// TIA Portal V17 export
// export: Created 2023-02-13T11:16:34.9023013Z, ExportSetting WithDefaults, DisplayName Totally Integrated Automation Portal, DisplayVersion V17, DisplayName TIA Portal Openness, DisplayVersion V17, DisplayName TIA Portal Teamcenter Gateway, DisplayVersion V17, DisplayName TIA Portal Version Control Interface, DisplayVersion V17, DisplayName SINAMICS Startdrive Advanced, DisplayVersion V17, DisplayName SINAMICS Startdrive G130, G150, S120, S150, SINAMICS MV, S210, DisplayVersion V17, DisplayName SINAMICS Startdrive G110M, G120, G120C, G120D, G120P, G115D, DisplayVersion V17, DisplayName STEP 7 Professional, DisplayVersion V17, DisplayName STEP 7 Safety, DisplayVersion V17, DisplayName WinCC Professional, DisplayVersion V17
FUNCTION_BLOCK "IO_Valve_Buffer"   // FB19, LAD
{ S7_Optimized_Access := 'FALSE' }
VERSION : 0.1
// stored: AutoNumber true, IsIECCheckEnabled false, SetENOAutomatically false, UDAEnableTagReadback false
   VAR_INPUT
      "lock 1" : Bool;
      "lock 2" : Bool;
      "lock 3" : Bool;
      "lock 4" : Bool;
      init : Bool;
      reset : Bool;
      testing : Bool;
   END_VAR
   VAR
      "AV-22.11" : "Valve";
      "AV-22.21" : "Valve";
      "AV-22.22" : "Valve";
      "AV-22.23" : "Valve";
      "AV-32.01" : "Valve";
      "AV-32.02" : "Valve";
      "AV-32.03" : "Valve";
      "AV-32.04" : "Valve";
      "AV-32.11" : "Valve";
      "AV-32.21" : "Valve";
      "AV-32.22" : "Valve";
      "AV-32.23" : "Valve";
      "AV-61.01" : "Valve";
      "AV-61.02" : "Valve";
      "AV-61.03" : "Valve";
      "AV-61.04" : "Valve";
      "AV-61.05" : "Valve";
      "AV-61.21" : "Valve";
      "AV-62.06" : "Valve";
      "AV-64.01" : "Valve";
      "AV-64.02" : "Valve";
      "AV-64.03" : "Valve";
      "AV-64.04" : "Valve";
      "AV-64.05" : "Valve";
      "AV-64.06" : "Valve";
      "AV-65.01" : "Valve";
      "AV-65.02" : "Valve";
      "AV-65.03" : "Valve";
      "AV-65.04" : "Valve";
      "AV-65.05" : "Valve";
      "AV-65.21" : "Valve";
      "AV-66.01" : "Valve";
      "AV-66.02" : "Valve";
      "AV-66.03" : "Valve";
      "AV-66.04" : "Valve";
      "AV-66.05" : "Valve";
      "AV-66.06" : "Valve";
      "AV-67.01" : "Valve";
      "AV-67.02" : "Valve";
      "AV-67.03" : "Valve";
      "AV-67.04" : "Valve";
      "AV-67.05" : "Valve";
      "AV-68.01" : "Valve";
      "AV-68.02" : "Valve";
      "AV-68.03" : "Valve";
      "AV-68.04" : "Valve";
      "AV-68.05" : "Valve";
      "AV-68.06" : "Valve";
   END_VAR
BEGIN

REGION Network 1 (SCL): FB OPEN AND CLOSE VALVE T-22
   IF #testing THEN
       // Statement section IF
       #"AV-22.11".FB_OPEN := #"AV-22.11".QCMD_OP;
       #"AV-22.11".FB_CLOSE := NOT #"AV-22.11".QCMD_OP;
       #"AV-22.21".FB_OPEN := #"AV-22.21".QCMD_OP;
       #"AV-22.21".FB_CLOSE := NOT #"AV-22.21".QCMD_OP;
       #"AV-22.22".FB_OPEN := #"AV-22.22".QCMD_OP;
       #"AV-22.22".FB_CLOSE := NOT #"AV-22.22".QCMD_OP;
       #"AV-22.23".FB_OPEN := #"AV-22.23".QCMD_OP;
       #"AV-22.23".FB_CLOSE := NOT #"AV-22.23".QCMD_OP;
   ELSE
       // Statement section ELSE
       #"AV-22.11".FB_OPEN := #"AV-22.11".QCMD_OP;
       #"AV-22.11".FB_CLOSE := NOT #"AV-22.11".QCMD_OP;
       #"AV-22.21".FB_OPEN := #"AV-22.21".QCMD_OP;
       #"AV-22.21".FB_CLOSE := NOT #"AV-22.21".QCMD_OP;
       #"AV-22.22".FB_OPEN := #"AV-22.22".QCMD_OP;
       #"AV-22.22".FB_CLOSE := NOT #"AV-22.22".QCMD_OP;
       #"AV-22.23".FB_OPEN := #"AV-22.23".QCMD_OP;
       #"AV-22.23".FB_CLOSE := NOT #"AV-22.23".QCMD_OP;
   END_IF;
END_REGION

NETWORK
TITLE = FB MONITORING TIME VALVE T-22
// FB OPEN TIME
      L     T#20s;
      T     #"AV-22.11".MON_T;
      T     #"AV-22.21".MON_T;
      T     #"AV-22.22".MON_T;
      T     #"AV-22.23".MON_T;
// FB CLOSE TIME
      L     T#20s;
      T     #"AV-22.11".MON_T_CLOSE;
      T     #"AV-22.21".MON_T_CLOSE;
      T     #"AV-22.22".MON_T_CLOSE;
      T     #"AV-22.23".MON_T_CLOSE;


REGION Network 3: AV-22.11
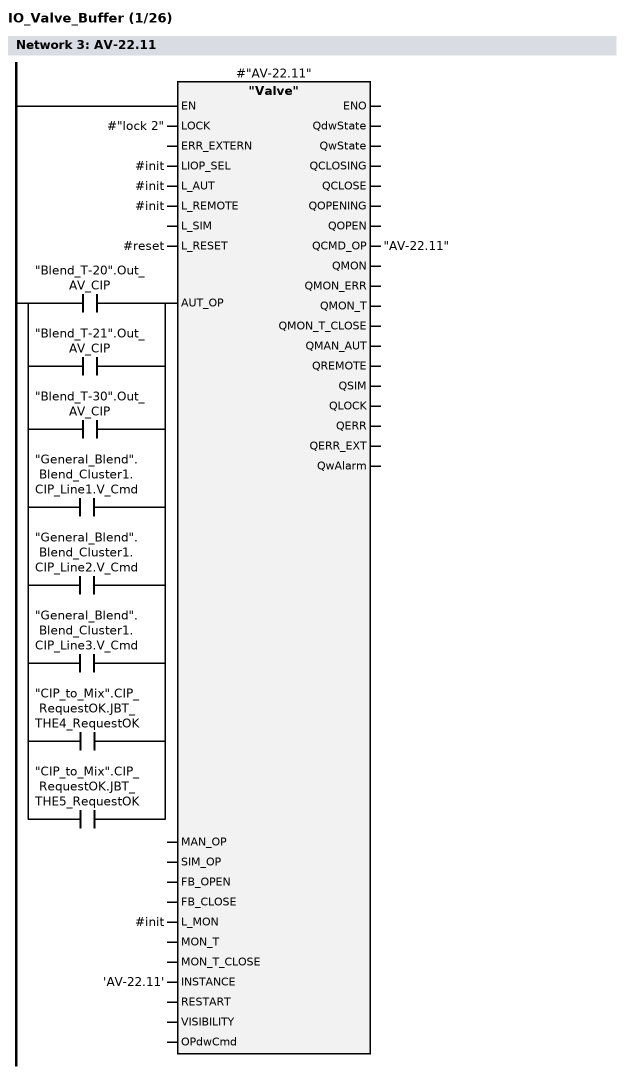
   RUNG wire#powerrail
      #"AV-22.11"(AUT_OP := wire#w1, LOCK := #"lock 2", ERR_EXTERN :=, LIOP_SEL := #init, L_AUT := #init, L_REMOTE := #init, L_SIM :=, L_RESET := #reset, MAN_OP :=, SIM_OP :=, FB_OPEN :=, FB_CLOSE :=, L_MON := #init, MON_T :=, MON_T_CLOSE :=, INSTANCE := 'AV-22.11', RESTART :=, VISIBILITY :=, OPdwCmd :=, QdwState =>, QwState =>, QCLOSING =>, QCLOSE =>, QOPENING =>, QOPEN =>, QCMD_OP => "AV-22.11", QMON =>, QMON_ERR =>, QMON_T =>, QMON_T_CLOSE =>, QMAN_AUT =>, QREMOTE =>, QSIM =>, QLOCK =>, QERR =>, QERR_EXT =>, QwAlarm =>)
   END_RUNG
   RUNG wire#powerrail
      Contact( "Blend_T-20".Out_AV_CIP )
   END_RUNG wire#w1
   RUNG wire#powerrail
      Contact( "Blend_T-21".Out_AV_CIP )
   END_RUNG wire#w1
   RUNG wire#powerrail
      Contact( "Blend_T-30".Out_AV_CIP )
   END_RUNG wire#w1
   RUNG wire#powerrail
      Contact( "General_Blend".Blend_Cluster1.CIP_Line1.V_Cmd )
   END_RUNG wire#w1
   RUNG wire#powerrail
      Contact( "General_Blend".Blend_Cluster1.CIP_Line2.V_Cmd )
   END_RUNG wire#w1
   RUNG wire#powerrail
      Contact( "General_Blend".Blend_Cluster1.CIP_Line3.V_Cmd )
   END_RUNG wire#w1
   RUNG wire#powerrail
      Contact( "CIP_to_Mix".CIP_RequestOK.JBT_THE4_RequestOK )
   END_RUNG wire#w1
   RUNG wire#powerrail
      Contact( "CIP_to_Mix".CIP_RequestOK.JBT_THE5_RequestOK )
   END_RUNG wire#w1
   // the same network as SCL:
   #"AV-22.11"(LOCK := #"lock 2",   // "Valve"
               LIOP_SEL := #init,
               L_AUT := #init,
               L_REMOTE := #init,
               L_RESET := #reset,
               AUT_OP := "Blend_T-20".Out_AV_CIP OR "Blend_T-21".Out_AV_CIP OR "Blend_T-30".Out_AV_CIP OR "General_Blend".Blend_Cluster1.CIP_Line1.V_Cmd OR "General_Blend".Blend_Cluster1.CIP_Line2.V_Cmd OR "General_Blend".Blend_Cluster1.CIP_Line3.V_Cmd OR "CIP_to_Mix".CIP_RequestOK.JBT_THE4_RequestOK OR "CIP_to_Mix".CIP_RequestOK.JBT_THE5_RequestOK,
               L_MON := #init,
               INSTANCE := 'AV-22.11',
               QCMD_OP => "AV-22.11");
END_REGION

REGION Network 4: AV-22.21
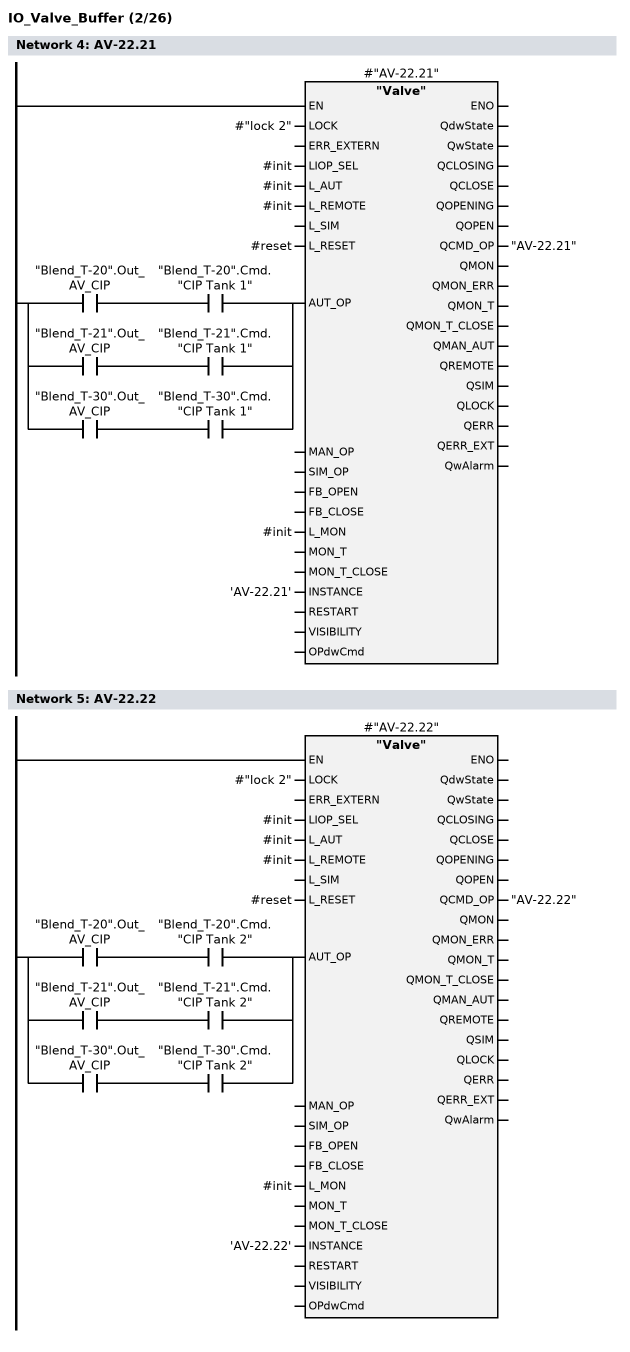
   RUNG wire#powerrail
      #"AV-22.21"(AUT_OP := wire#w1, LOCK := #"lock 2", ERR_EXTERN :=, LIOP_SEL := #init, L_AUT := #init, L_REMOTE := #init, L_SIM :=, L_RESET := #reset, MAN_OP :=, SIM_OP :=, FB_OPEN :=, FB_CLOSE :=, L_MON := #init, MON_T :=, MON_T_CLOSE :=, INSTANCE := 'AV-22.21', RESTART :=, VISIBILITY :=, OPdwCmd :=, QdwState =>, QwState =>, QCLOSING =>, QCLOSE =>, QOPENING =>, QOPEN =>, QCMD_OP => "AV-22.21", QMON =>, QMON_ERR =>, QMON_T =>, QMON_T_CLOSE =>, QMAN_AUT =>, QREMOTE =>, QSIM =>, QLOCK =>, QERR =>, QERR_EXT =>, QwAlarm =>)
   END_RUNG
   RUNG wire#powerrail
      Contact( "Blend_T-20".Out_AV_CIP )
      Contact( "Blend_T-20".Cmd."CIP Tank 1" )
   END_RUNG wire#w1
   RUNG wire#powerrail
      Contact( "Blend_T-21".Out_AV_CIP )
      Contact( "Blend_T-21".Cmd."CIP Tank 1" )
   END_RUNG wire#w1
   RUNG wire#powerrail
      Contact( "Blend_T-30".Out_AV_CIP )
      Contact( "Blend_T-30".Cmd."CIP Tank 1" )
   END_RUNG wire#w1
   // the same network as SCL:
   #"AV-22.21"(LOCK := #"lock 2",   // "Valve"
               LIOP_SEL := #init,
               L_AUT := #init,
               L_REMOTE := #init,
               L_RESET := #reset,
               AUT_OP := ("Blend_T-20".Out_AV_CIP AND "Blend_T-20".Cmd."CIP Tank 1") OR ("Blend_T-21".Out_AV_CIP AND "Blend_T-21".Cmd."CIP Tank 1") OR ("Blend_T-30".Out_AV_CIP AND "Blend_T-30".Cmd."CIP Tank 1"),
               L_MON := #init,
               INSTANCE := 'AV-22.21',
               QCMD_OP => "AV-22.21");
END_REGION

REGION Network 5: AV-22.22
   RUNG wire#powerrail
      #"AV-22.22"(AUT_OP := wire#w1, LOCK := #"lock 2", ERR_EXTERN :=, LIOP_SEL := #init, L_AUT := #init, L_REMOTE := #init, L_SIM :=, L_RESET := #reset, MAN_OP :=, SIM_OP :=, FB_OPEN :=, FB_CLOSE :=, L_MON := #init, MON_T :=, MON_T_CLOSE :=, INSTANCE := 'AV-22.22', RESTART :=, VISIBILITY :=, OPdwCmd :=, QdwState =>, QwState =>, QCLOSING =>, QCLOSE =>, QOPENING =>, QOPEN =>, QCMD_OP => "AV-22.22", QMON =>, QMON_ERR =>, QMON_T =>, QMON_T_CLOSE =>, QMAN_AUT =>, QREMOTE =>, QSIM =>, QLOCK =>, QERR =>, QERR_EXT =>, QwAlarm =>)
   END_RUNG
   RUNG wire#powerrail
      Contact( "Blend_T-20".Out_AV_CIP )
      Contact( "Blend_T-20".Cmd."CIP Tank 2" )
   END_RUNG wire#w1
   RUNG wire#powerrail
      Contact( "Blend_T-21".Out_AV_CIP )
      Contact( "Blend_T-21".Cmd."CIP Tank 2" )
   END_RUNG wire#w1
   RUNG wire#powerrail
      Contact( "Blend_T-30".Out_AV_CIP )
      Contact( "Blend_T-30".Cmd."CIP Tank 2" )
   END_RUNG wire#w1
   // the same network as SCL:
   #"AV-22.22"(LOCK := #"lock 2",   // "Valve"
               LIOP_SEL := #init,
               L_AUT := #init,
               L_REMOTE := #init,
               L_RESET := #reset,
               AUT_OP := ("Blend_T-20".Out_AV_CIP AND "Blend_T-20".Cmd."CIP Tank 2") OR ("Blend_T-21".Out_AV_CIP AND "Blend_T-21".Cmd."CIP Tank 2") OR ("Blend_T-30".Out_AV_CIP AND "Blend_T-30".Cmd."CIP Tank 2"),
               L_MON := #init,
               INSTANCE := 'AV-22.22',
               QCMD_OP => "AV-22.22");
END_REGION

REGION Network 6: AV-22.23
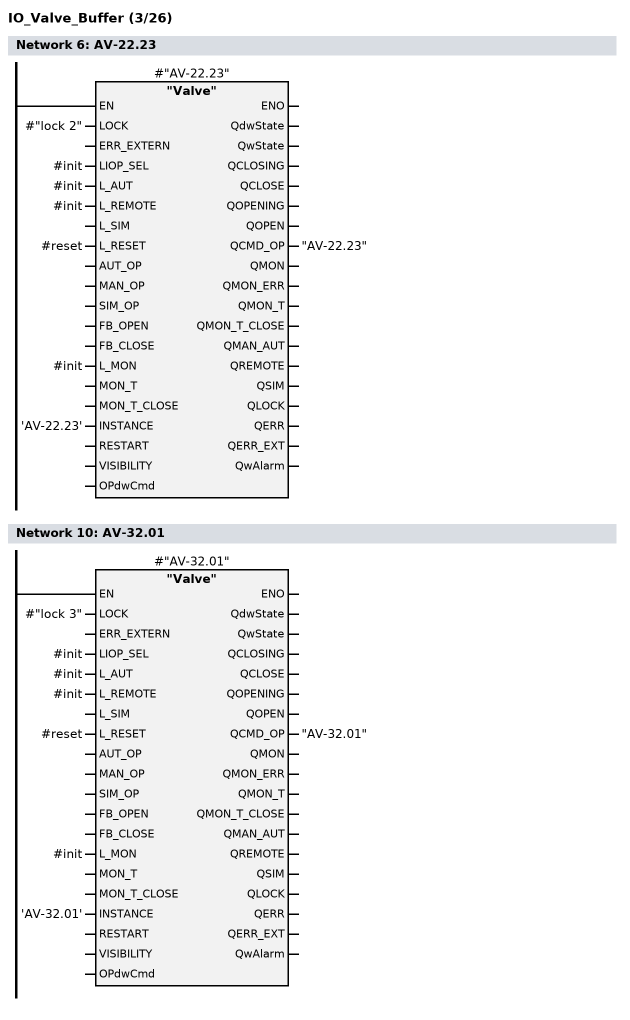
   RUNG wire#powerrail
      #"AV-22.23"(LOCK := #"lock 2", ERR_EXTERN :=, LIOP_SEL := #init, L_AUT := #init, L_REMOTE := #init, L_SIM :=, L_RESET := #reset, AUT_OP :=, MAN_OP :=, SIM_OP :=, FB_OPEN :=, FB_CLOSE :=, L_MON := #init, MON_T :=, MON_T_CLOSE :=, INSTANCE := 'AV-22.23', RESTART :=, VISIBILITY :=, OPdwCmd :=, QdwState =>, QwState =>, QCLOSING =>, QCLOSE =>, QOPENING =>, QOPEN =>, QCMD_OP => "AV-22.23", QMON =>, QMON_ERR =>, QMON_T =>, QMON_T_CLOSE =>, QMAN_AUT =>, QREMOTE =>, QSIM =>, QLOCK =>, QERR =>, QERR_EXT =>, QwAlarm =>)
   END_RUNG
   // the same network as SCL:
   #"AV-22.23"(LOCK := #"lock 2",   // "Valve"
               LIOP_SEL := #init,
               L_AUT := #init,
               L_REMOTE := #init,
               L_RESET := #reset,
               L_MON := #init,
               INSTANCE := 'AV-22.23',
               QCMD_OP => "AV-22.23");
END_REGION

REGION Network 8 (SCL): FB OPEN AND CLOSE VALVE T-32
   IF #testing THEN
       // Statement section IF
       #"AV-32.01".FB_OPEN := #"AV-32.01".QCMD_OP;
       #"AV-32.01".FB_CLOSE := NOT #"AV-32.01".QCMD_OP;
       #"AV-32.02".FB_OPEN := #"AV-32.02".QCMD_OP;
       #"AV-32.02".FB_CLOSE := NOT #"AV-32.02".QCMD_OP;
       #"AV-32.03".FB_OPEN := #"AV-32.03".QCMD_OP;
       #"AV-32.03".FB_CLOSE := NOT #"AV-32.03".QCMD_OP;
       #"AV-32.04".FB_OPEN := #"AV-32.04".QCMD_OP;
       #"AV-32.04".FB_CLOSE := NOT #"AV-32.04".QCMD_OP;
       #"AV-32.11".FB_OPEN := #"AV-32.11".QCMD_OP;
       #"AV-32.11".FB_CLOSE := NOT #"AV-32.11".QCMD_OP;
       #"AV-32.21".FB_OPEN := #"AV-32.21".QCMD_OP;
       #"AV-32.21".FB_CLOSE := NOT #"AV-32.21".QCMD_OP;
       #"AV-32.22".FB_OPEN := #"AV-32.22".QCMD_OP;
       #"AV-32.22".FB_CLOSE := NOT #"AV-32.22".QCMD_OP;
       #"AV-32.23".FB_OPEN := #"AV-32.23".QCMD_OP;
       #"AV-32.23".FB_CLOSE := NOT #"AV-32.23".QCMD_OP;
   ELSE
       // Statement section ELSE
       #"AV-32.01".FB_OPEN := #"AV-32.01".QCMD_OP;
       #"AV-32.01".FB_CLOSE := NOT #"AV-32.01".QCMD_OP;
       #"AV-32.02".FB_OPEN := #"AV-32.02".QCMD_OP;
       #"AV-32.02".FB_CLOSE := NOT #"AV-32.02".QCMD_OP;
       #"AV-32.03".FB_OPEN := #"AV-32.03".QCMD_OP;
       #"AV-32.03".FB_CLOSE := NOT #"AV-32.03".QCMD_OP;
       #"AV-32.04".FB_OPEN := #"AV-32.04".QCMD_OP;
       #"AV-32.04".FB_CLOSE := NOT #"AV-32.04".QCMD_OP;
       #"AV-32.11".FB_OPEN := #"AV-32.11".QCMD_OP;
       #"AV-32.11".FB_CLOSE := NOT #"AV-32.11".QCMD_OP;
       #"AV-32.21".FB_OPEN := #"AV-32.21".QCMD_OP;
       #"AV-32.21".FB_CLOSE := NOT #"AV-32.21".QCMD_OP;
       #"AV-32.22".FB_OPEN := #"AV-32.22".QCMD_OP;
       #"AV-32.22".FB_CLOSE := NOT #"AV-32.22".QCMD_OP;
       #"AV-32.23".FB_OPEN := #"AV-32.23".QCMD_OP;
       #"AV-32.23".FB_CLOSE := NOT #"AV-32.23".QCMD_OP;
   END_IF;
END_REGION

NETWORK
TITLE = FB MONITORING TIME VALVE T-32
// FB OPEN TIME
      L     T#20s;
      T     #"AV-32.01".MON_T;
      T     #"AV-32.02".MON_T;
      T     #"AV-32.03".MON_T;
      T     #"AV-32.04".MON_T;
      T     #"AV-32.11".MON_T;
      T     #"AV-32.21".MON_T;
      T     #"AV-32.22".MON_T;
      T     #"AV-32.23".MON_T;
// FB CLOSE TIME
      L     T#20s;
      T     #"AV-32.01".MON_T_CLOSE;
      T     #"AV-32.02".MON_T_CLOSE;
      T     #"AV-32.03".MON_T_CLOSE;
      T     #"AV-32.04".MON_T_CLOSE;
      T     #"AV-32.11".MON_T_CLOSE;
      T     #"AV-32.21".MON_T_CLOSE;
      T     #"AV-32.22".MON_T_CLOSE;
      T     #"AV-32.23".MON_T_CLOSE;


REGION Network 10: AV-32.01
   RUNG wire#powerrail
      #"AV-32.01"(LOCK := #"lock 3", ERR_EXTERN :=, LIOP_SEL := #init, L_AUT := #init, L_REMOTE := #init, L_SIM :=, L_RESET := #reset, AUT_OP :=, MAN_OP :=, SIM_OP :=, FB_OPEN :=, FB_CLOSE :=, L_MON := #init, MON_T :=, MON_T_CLOSE :=, INSTANCE := 'AV-32.01', RESTART :=, VISIBILITY :=, OPdwCmd :=, QdwState =>, QwState =>, QCLOSING =>, QCLOSE =>, QOPENING =>, QOPEN =>, QCMD_OP => "AV-32.01", QMON =>, QMON_ERR =>, QMON_T =>, QMON_T_CLOSE =>, QMAN_AUT =>, QREMOTE =>, QSIM =>, QLOCK =>, QERR =>, QERR_EXT =>, QwAlarm =>)
   END_RUNG
   // the same network as SCL:
   #"AV-32.01"(LOCK := #"lock 3",   // "Valve"
               LIOP_SEL := #init,
               L_AUT := #init,
               L_REMOTE := #init,
               L_RESET := #reset,
               L_MON := #init,
               INSTANCE := 'AV-32.01',
               QCMD_OP => "AV-32.01");
END_REGION

REGION Network 11: AV-32.02
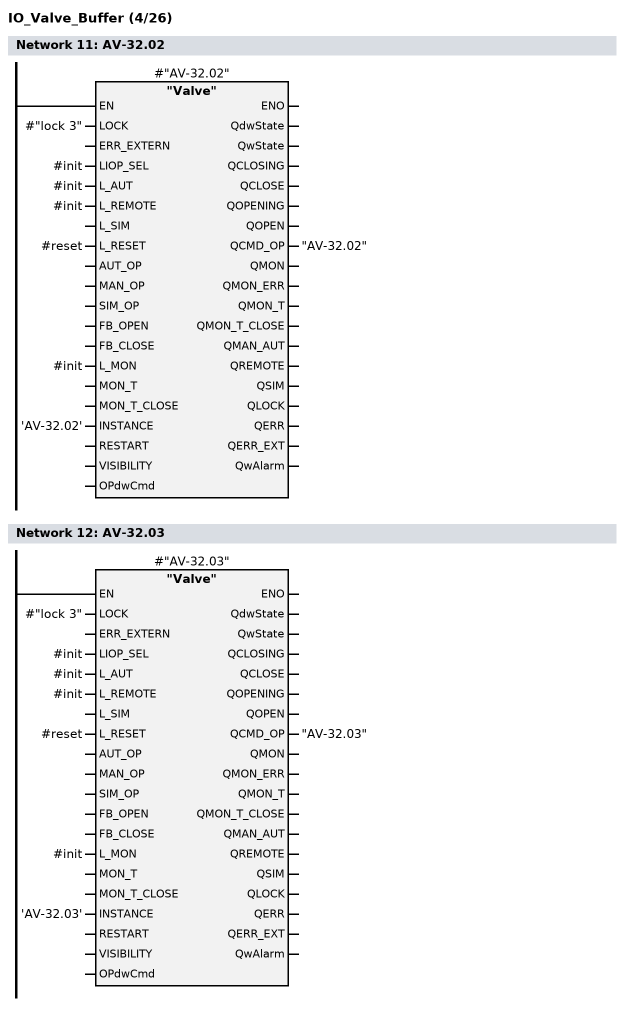
   RUNG wire#powerrail
      #"AV-32.02"(LOCK := #"lock 3", ERR_EXTERN :=, LIOP_SEL := #init, L_AUT := #init, L_REMOTE := #init, L_SIM :=, L_RESET := #reset, AUT_OP :=, MAN_OP :=, SIM_OP :=, FB_OPEN :=, FB_CLOSE :=, L_MON := #init, MON_T :=, MON_T_CLOSE :=, INSTANCE := 'AV-32.02', RESTART :=, VISIBILITY :=, OPdwCmd :=, QdwState =>, QwState =>, QCLOSING =>, QCLOSE =>, QOPENING =>, QOPEN =>, QCMD_OP => "AV-32.02", QMON =>, QMON_ERR =>, QMON_T =>, QMON_T_CLOSE =>, QMAN_AUT =>, QREMOTE =>, QSIM =>, QLOCK =>, QERR =>, QERR_EXT =>, QwAlarm =>)
   END_RUNG
   // the same network as SCL:
   #"AV-32.02"(LOCK := #"lock 3",   // "Valve"
               LIOP_SEL := #init,
               L_AUT := #init,
               L_REMOTE := #init,
               L_RESET := #reset,
               L_MON := #init,
               INSTANCE := 'AV-32.02',
               QCMD_OP => "AV-32.02");
END_REGION

REGION Network 12: AV-32.03
   RUNG wire#powerrail
      #"AV-32.03"(LOCK := #"lock 3", ERR_EXTERN :=, LIOP_SEL := #init, L_AUT := #init, L_REMOTE := #init, L_SIM :=, L_RESET := #reset, AUT_OP :=, MAN_OP :=, SIM_OP :=, FB_OPEN :=, FB_CLOSE :=, L_MON := #init, MON_T :=, MON_T_CLOSE :=, INSTANCE := 'AV-32.03', RESTART :=, VISIBILITY :=, OPdwCmd :=, QdwState =>, QwState =>, QCLOSING =>, QCLOSE =>, QOPENING =>, QOPEN =>, QCMD_OP => "AV-32.03", QMON =>, QMON_ERR =>, QMON_T =>, QMON_T_CLOSE =>, QMAN_AUT =>, QREMOTE =>, QSIM =>, QLOCK =>, QERR =>, QERR_EXT =>, QwAlarm =>)
   END_RUNG
   // the same network as SCL:
   #"AV-32.03"(LOCK := #"lock 3",   // "Valve"
               LIOP_SEL := #init,
               L_AUT := #init,
               L_REMOTE := #init,
               L_RESET := #reset,
               L_MON := #init,
               INSTANCE := 'AV-32.03',
               QCMD_OP => "AV-32.03");
END_REGION

REGION Network 13: AV-32.04
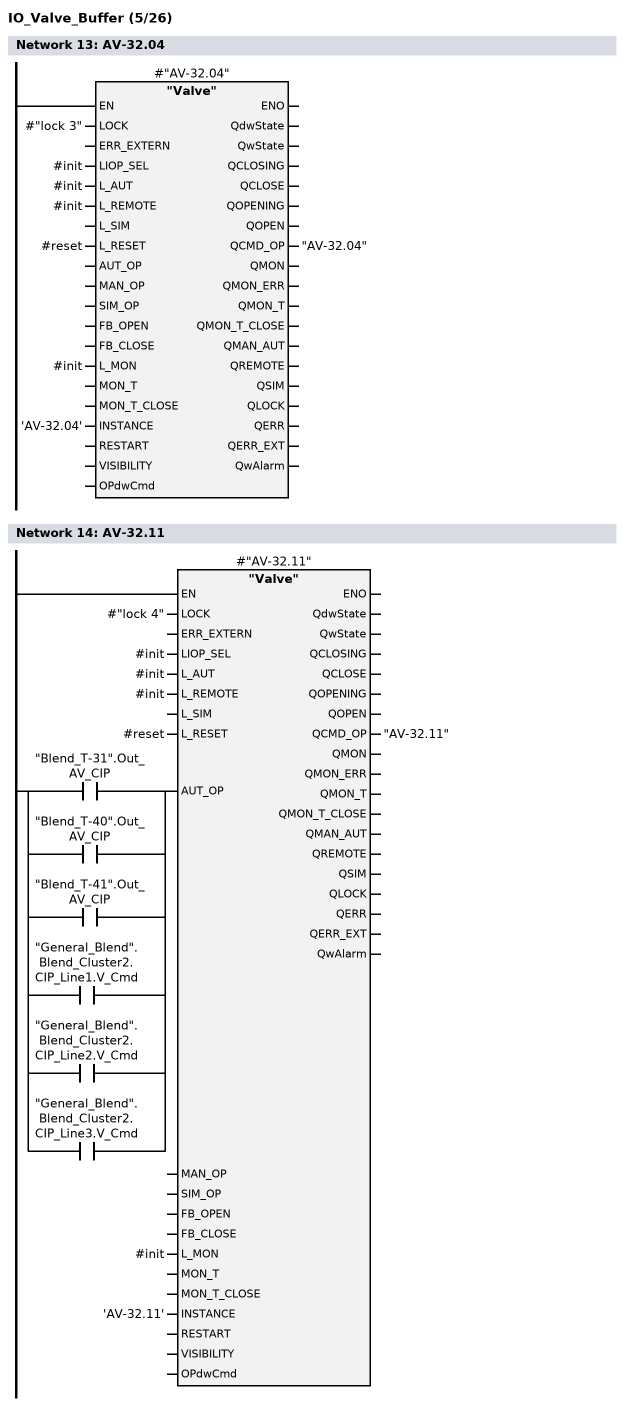
   RUNG wire#powerrail
      #"AV-32.04"(LOCK := #"lock 3", ERR_EXTERN :=, LIOP_SEL := #init, L_AUT := #init, L_REMOTE := #init, L_SIM :=, L_RESET := #reset, AUT_OP :=, MAN_OP :=, SIM_OP :=, FB_OPEN :=, FB_CLOSE :=, L_MON := #init, MON_T :=, MON_T_CLOSE :=, INSTANCE := 'AV-32.04', RESTART :=, VISIBILITY :=, OPdwCmd :=, QdwState =>, QwState =>, QCLOSING =>, QCLOSE =>, QOPENING =>, QOPEN =>, QCMD_OP => "AV-32.04", QMON =>, QMON_ERR =>, QMON_T =>, QMON_T_CLOSE =>, QMAN_AUT =>, QREMOTE =>, QSIM =>, QLOCK =>, QERR =>, QERR_EXT =>, QwAlarm =>)
   END_RUNG
   // the same network as SCL:
   #"AV-32.04"(LOCK := #"lock 3",   // "Valve"
               LIOP_SEL := #init,
               L_AUT := #init,
               L_REMOTE := #init,
               L_RESET := #reset,
               L_MON := #init,
               INSTANCE := 'AV-32.04',
               QCMD_OP => "AV-32.04");
END_REGION

REGION Network 14: AV-32.11
   RUNG wire#powerrail
      #"AV-32.11"(AUT_OP := wire#w1, LOCK := #"lock 4", ERR_EXTERN :=, LIOP_SEL := #init, L_AUT := #init, L_REMOTE := #init, L_SIM :=, L_RESET := #reset, MAN_OP :=, SIM_OP :=, FB_OPEN :=, FB_CLOSE :=, L_MON := #init, MON_T :=, MON_T_CLOSE :=, INSTANCE := 'AV-32.11', RESTART :=, VISIBILITY :=, OPdwCmd :=, QdwState =>, QwState =>, QCLOSING =>, QCLOSE =>, QOPENING =>, QOPEN =>, QCMD_OP => "AV-32.11", QMON =>, QMON_ERR =>, QMON_T =>, QMON_T_CLOSE =>, QMAN_AUT =>, QREMOTE =>, QSIM =>, QLOCK =>, QERR =>, QERR_EXT =>, QwAlarm =>)
   END_RUNG
   RUNG wire#powerrail
      Contact( "Blend_T-31".Out_AV_CIP )
   END_RUNG wire#w1
   RUNG wire#powerrail
      Contact( "Blend_T-40".Out_AV_CIP )
   END_RUNG wire#w1
   RUNG wire#powerrail
      Contact( "Blend_T-41".Out_AV_CIP )
   END_RUNG wire#w1
   RUNG wire#powerrail
      Contact( "General_Blend".Blend_Cluster2.CIP_Line1.V_Cmd )
   END_RUNG wire#w1
   RUNG wire#powerrail
      Contact( "General_Blend".Blend_Cluster2.CIP_Line2.V_Cmd )
   END_RUNG wire#w1
   RUNG wire#powerrail
      Contact( "General_Blend".Blend_Cluster2.CIP_Line3.V_Cmd )
   END_RUNG wire#w1
   // the same network as SCL:
   #"AV-32.11"(LOCK := #"lock 4",   // "Valve"
               LIOP_SEL := #init,
               L_AUT := #init,
               L_REMOTE := #init,
               L_RESET := #reset,
               AUT_OP := "Blend_T-31".Out_AV_CIP OR "Blend_T-40".Out_AV_CIP OR "Blend_T-41".Out_AV_CIP OR "General_Blend".Blend_Cluster2.CIP_Line1.V_Cmd OR "General_Blend".Blend_Cluster2.CIP_Line2.V_Cmd OR "General_Blend".Blend_Cluster2.CIP_Line3.V_Cmd,
               L_MON := #init,
               INSTANCE := 'AV-32.11',
               QCMD_OP => "AV-32.11");
END_REGION

REGION Network 15: AV-32.21
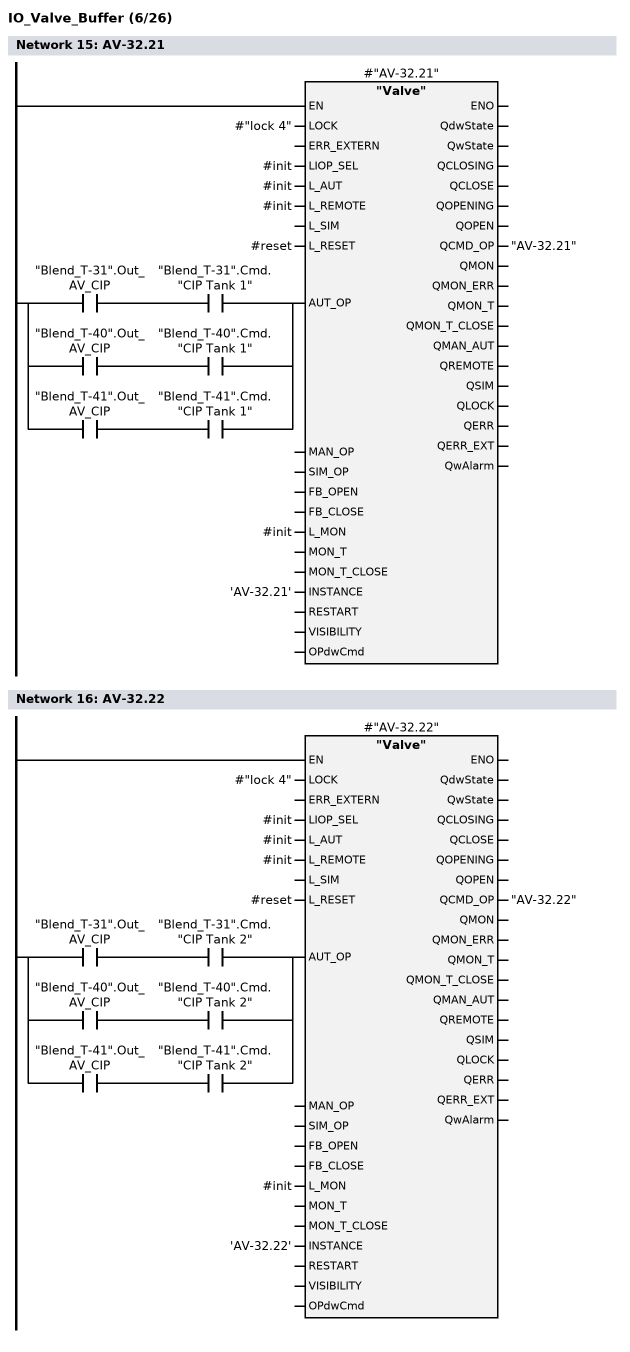
   RUNG wire#powerrail
      #"AV-32.21"(AUT_OP := wire#w1, LOCK := #"lock 4", ERR_EXTERN :=, LIOP_SEL := #init, L_AUT := #init, L_REMOTE := #init, L_SIM :=, L_RESET := #reset, MAN_OP :=, SIM_OP :=, FB_OPEN :=, FB_CLOSE :=, L_MON := #init, MON_T :=, MON_T_CLOSE :=, INSTANCE := 'AV-32.21', RESTART :=, VISIBILITY :=, OPdwCmd :=, QdwState =>, QwState =>, QCLOSING =>, QCLOSE =>, QOPENING =>, QOPEN =>, QCMD_OP => "AV-32.21", QMON =>, QMON_ERR =>, QMON_T =>, QMON_T_CLOSE =>, QMAN_AUT =>, QREMOTE =>, QSIM =>, QLOCK =>, QERR =>, QERR_EXT =>, QwAlarm =>)
   END_RUNG
   RUNG wire#powerrail
      Contact( "Blend_T-31".Out_AV_CIP )
      Contact( "Blend_T-31".Cmd."CIP Tank 1" )
   END_RUNG wire#w1
   RUNG wire#powerrail
      Contact( "Blend_T-40".Out_AV_CIP )
      Contact( "Blend_T-40".Cmd."CIP Tank 1" )
   END_RUNG wire#w1
   RUNG wire#powerrail
      Contact( "Blend_T-41".Out_AV_CIP )
      Contact( "Blend_T-41".Cmd."CIP Tank 1" )
   END_RUNG wire#w1
   // the same network as SCL:
   #"AV-32.21"(LOCK := #"lock 4",   // "Valve"
               LIOP_SEL := #init,
               L_AUT := #init,
               L_REMOTE := #init,
               L_RESET := #reset,
               AUT_OP := ("Blend_T-31".Out_AV_CIP AND "Blend_T-31".Cmd."CIP Tank 1") OR ("Blend_T-40".Out_AV_CIP AND "Blend_T-40".Cmd."CIP Tank 1") OR ("Blend_T-41".Out_AV_CIP AND "Blend_T-41".Cmd."CIP Tank 1"),
               L_MON := #init,
               INSTANCE := 'AV-32.21',
               QCMD_OP => "AV-32.21");
END_REGION

REGION Network 16: AV-32.22
   RUNG wire#powerrail
      #"AV-32.22"(AUT_OP := wire#w1, LOCK := #"lock 4", ERR_EXTERN :=, LIOP_SEL := #init, L_AUT := #init, L_REMOTE := #init, L_SIM :=, L_RESET := #reset, MAN_OP :=, SIM_OP :=, FB_OPEN :=, FB_CLOSE :=, L_MON := #init, MON_T :=, MON_T_CLOSE :=, INSTANCE := 'AV-32.22', RESTART :=, VISIBILITY :=, OPdwCmd :=, QdwState =>, QwState =>, QCLOSING =>, QCLOSE =>, QOPENING =>, QOPEN =>, QCMD_OP => "AV-32.22", QMON =>, QMON_ERR =>, QMON_T =>, QMON_T_CLOSE =>, QMAN_AUT =>, QREMOTE =>, QSIM =>, QLOCK =>, QERR =>, QERR_EXT =>, QwAlarm =>)
   END_RUNG
   RUNG wire#powerrail
      Contact( "Blend_T-31".Out_AV_CIP )
      Contact( "Blend_T-31".Cmd."CIP Tank 2" )
   END_RUNG wire#w1
   RUNG wire#powerrail
      Contact( "Blend_T-40".Out_AV_CIP )
      Contact( "Blend_T-40".Cmd."CIP Tank 2" )
   END_RUNG wire#w1
   RUNG wire#powerrail
      Contact( "Blend_T-41".Out_AV_CIP )
      Contact( "Blend_T-41".Cmd."CIP Tank 2" )
   END_RUNG wire#w1
   // the same network as SCL:
   #"AV-32.22"(LOCK := #"lock 4",   // "Valve"
               LIOP_SEL := #init,
               L_AUT := #init,
               L_REMOTE := #init,
               L_RESET := #reset,
               AUT_OP := ("Blend_T-31".Out_AV_CIP AND "Blend_T-31".Cmd."CIP Tank 2") OR ("Blend_T-40".Out_AV_CIP AND "Blend_T-40".Cmd."CIP Tank 2") OR ("Blend_T-41".Out_AV_CIP AND "Blend_T-41".Cmd."CIP Tank 2"),
               L_MON := #init,
               INSTANCE := 'AV-32.22',
               QCMD_OP => "AV-32.22");
END_REGION

REGION Network 17: AV-32.23
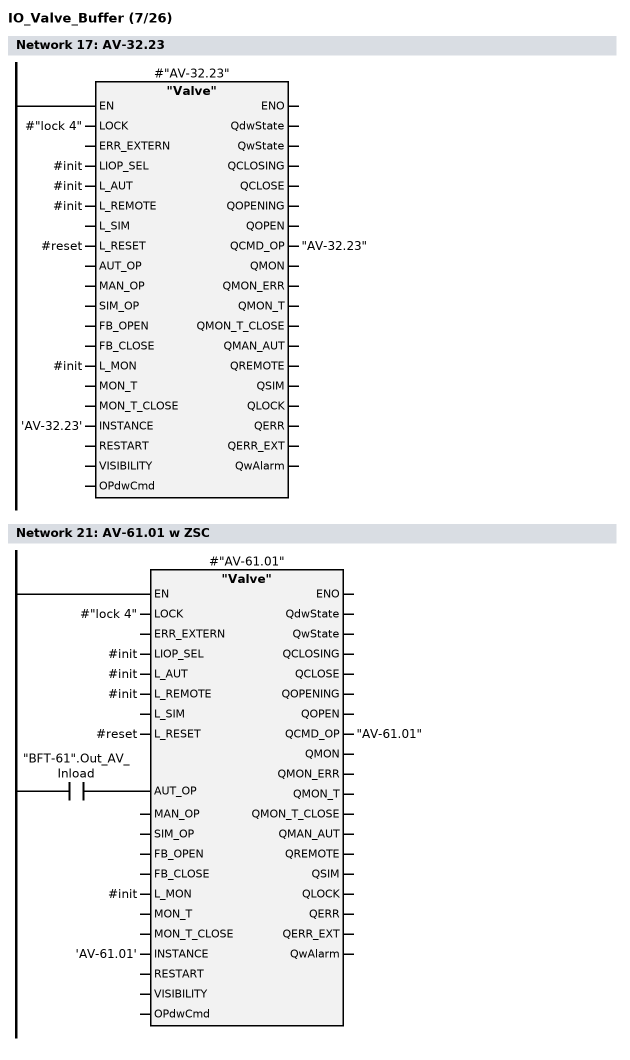
   RUNG wire#powerrail
      #"AV-32.23"(LOCK := #"lock 4", ERR_EXTERN :=, LIOP_SEL := #init, L_AUT := #init, L_REMOTE := #init, L_SIM :=, L_RESET := #reset, AUT_OP :=, MAN_OP :=, SIM_OP :=, FB_OPEN :=, FB_CLOSE :=, L_MON := #init, MON_T :=, MON_T_CLOSE :=, INSTANCE := 'AV-32.23', RESTART :=, VISIBILITY :=, OPdwCmd :=, QdwState =>, QwState =>, QCLOSING =>, QCLOSE =>, QOPENING =>, QOPEN =>, QCMD_OP => "AV-32.23", QMON =>, QMON_ERR =>, QMON_T =>, QMON_T_CLOSE =>, QMAN_AUT =>, QREMOTE =>, QSIM =>, QLOCK =>, QERR =>, QERR_EXT =>, QwAlarm =>)
   END_RUNG
   // the same network as SCL:
   #"AV-32.23"(LOCK := #"lock 4",   // "Valve"
               LIOP_SEL := #init,
               L_AUT := #init,
               L_REMOTE := #init,
               L_RESET := #reset,
               L_MON := #init,
               INSTANCE := 'AV-32.23',
               QCMD_OP => "AV-32.23");
END_REGION

REGION Network 19 (SCL): FB OPEN AND CLOSE VALVE T-61
   IF #testing THEN
       // Statement section IF
       #"AV-61.01".FB_OPEN := #"AV-61.01".QCMD_OP;
       #"AV-61.01".FB_CLOSE := NOT #"AV-61.01".QCMD_OP;
       #"AV-61.02".FB_OPEN := #"AV-61.02".QCMD_OP;
       #"AV-61.02".FB_CLOSE := NOT #"AV-61.02".QCMD_OP;
       #"AV-61.03".FB_OPEN := #"AV-61.03".QCMD_OP;
       #"AV-61.03".FB_CLOSE := NOT #"AV-61.03".QCMD_OP;
       #"AV-61.04".FB_OPEN := #"AV-61.04".QCMD_OP;
       #"AV-61.04".FB_CLOSE := NOT #"AV-61.04".QCMD_OP;
       #"AV-61.05".FB_OPEN := #"AV-61.05".QCMD_OP;
       #"AV-61.05".FB_CLOSE := NOT #"AV-61.05".QCMD_OP;
       #"AV-61.21".FB_OPEN := #"AV-61.21".QCMD_OP;
       #"AV-61.21".FB_CLOSE := NOT #"AV-61.21".QCMD_OP;
   ELSE
       // Statement section ELSE
       #"AV-61.01".FB_OPEN := NOT "ZSC-61.01";
       #"AV-61.01".FB_CLOSE := "ZSC-61.01";
       #"AV-61.02".FB_OPEN := #"AV-61.02".QCMD_OP;
       #"AV-61.02".FB_CLOSE := NOT #"AV-61.02".QCMD_OP;
       #"AV-61.03".FB_OPEN := NOT "ZSC-61.03";
       #"AV-61.03".FB_CLOSE := "ZSC-61.03";
       #"AV-61.04".FB_OPEN := #"AV-61.04".QCMD_OP;
       #"AV-61.04".FB_CLOSE := NOT #"AV-61.04".QCMD_OP;
       #"AV-61.05".FB_OPEN := #"AV-61.05".QCMD_OP;
       #"AV-61.05".FB_CLOSE := NOT #"AV-61.05".QCMD_OP;
       #"AV-61.21".FB_OPEN := #"AV-61.21".QCMD_OP;
       #"AV-61.21".FB_CLOSE := NOT #"AV-61.21".QCMD_OP;
   END_IF;
END_REGION

NETWORK
TITLE = FB MONITORING TIME VALVE T-61
// FB OPEN TIME
      L     T#20s;
      T     #"AV-61.01".MON_T;
      T     #"AV-61.02".MON_T;
      T     #"AV-61.03".MON_T;
      T     #"AV-61.04".MON_T;
      T     #"AV-61.05".MON_T;
      T     #"AV-61.21".MON_T;
// FB CLOSE TIME
      L     T#20s;
      T     #"AV-61.01".MON_T_CLOSE;
      T     #"AV-61.02".MON_T_CLOSE;
      T     #"AV-61.03".MON_T_CLOSE;
      T     #"AV-61.04".MON_T_CLOSE;
      T     #"AV-61.05".MON_T_CLOSE;
      T     #"AV-61.21".MON_T_CLOSE;

REGION Network 21: AV-61.01 w ZSC
   RUNG wire#powerrail
      #"AV-61.01"(AUT_OP := wire#w1, LOCK := #"lock 4", ERR_EXTERN :=, LIOP_SEL := #init, L_AUT := #init, L_REMOTE := #init, L_SIM :=, L_RESET := #reset, MAN_OP :=, SIM_OP :=, FB_OPEN :=, FB_CLOSE :=, L_MON := #init, MON_T :=, MON_T_CLOSE :=, INSTANCE := 'AV-61.01', RESTART :=, VISIBILITY :=, OPdwCmd :=, QdwState =>, QwState =>, QCLOSING =>, QCLOSE =>, QOPENING =>, QOPEN =>, QCMD_OP => "AV-61.01", QMON =>, QMON_ERR =>, QMON_T =>, QMON_T_CLOSE =>, QMAN_AUT =>, QREMOTE =>, QSIM =>, QLOCK =>, QERR =>, QERR_EXT =>, QwAlarm =>)
   END_RUNG
   RUNG wire#powerrail
      Contact( "BFT-61".Out_AV_Inload )
   END_RUNG wire#w1
   // the same network as SCL:
   #"AV-61.01"(LOCK := #"lock 4",   // "Valve"
               LIOP_SEL := #init,
               L_AUT := #init,
               L_REMOTE := #init,
               L_RESET := #reset,
               AUT_OP := "BFT-61".Out_AV_Inload,
               L_MON := #init,
               INSTANCE := 'AV-61.01',
               QCMD_OP => "AV-61.01");
END_REGION

REGION Network 22: AV-61.02
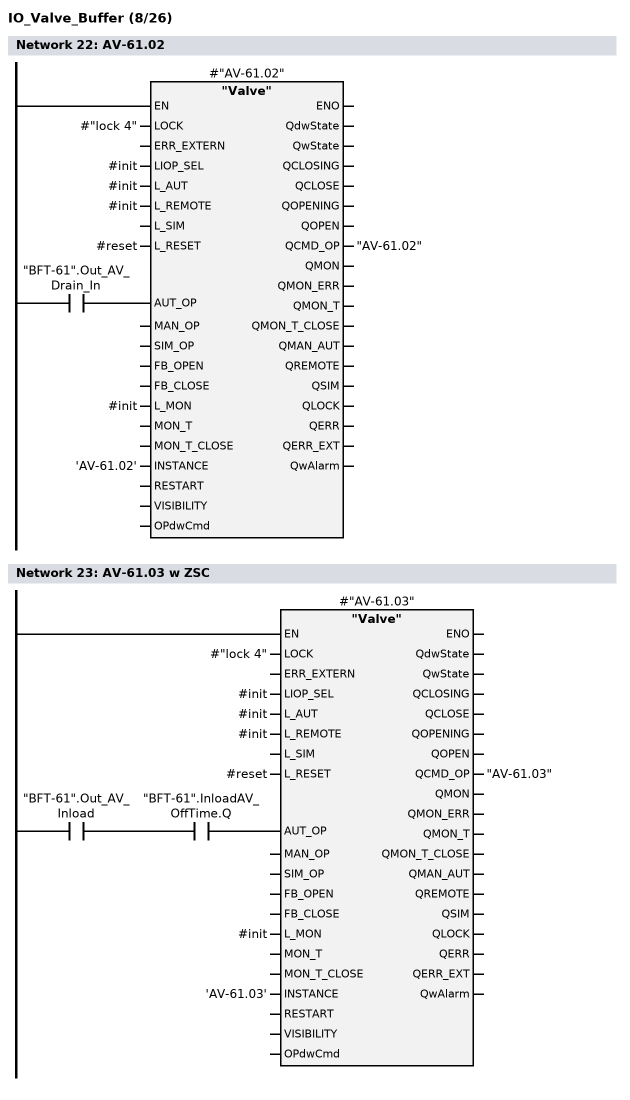
   RUNG wire#powerrail
      #"AV-61.02"(AUT_OP := wire#w1, LOCK := #"lock 4", ERR_EXTERN :=, LIOP_SEL := #init, L_AUT := #init, L_REMOTE := #init, L_SIM :=, L_RESET := #reset, MAN_OP :=, SIM_OP :=, FB_OPEN :=, FB_CLOSE :=, L_MON := #init, MON_T :=, MON_T_CLOSE :=, INSTANCE := 'AV-61.02', RESTART :=, VISIBILITY :=, OPdwCmd :=, QdwState =>, QwState =>, QCLOSING =>, QCLOSE =>, QOPENING =>, QOPEN =>, QCMD_OP => "AV-61.02", QMON =>, QMON_ERR =>, QMON_T =>, QMON_T_CLOSE =>, QMAN_AUT =>, QREMOTE =>, QSIM =>, QLOCK =>, QERR =>, QERR_EXT =>, QwAlarm =>)
   END_RUNG
   RUNG wire#powerrail
      Contact( "BFT-61".Out_AV_Drain_In )
   END_RUNG wire#w1
   // the same network as SCL:
   #"AV-61.02"(LOCK := #"lock 4",   // "Valve"
               LIOP_SEL := #init,
               L_AUT := #init,
               L_REMOTE := #init,
               L_RESET := #reset,
               AUT_OP := "BFT-61".Out_AV_Drain_In,
               L_MON := #init,
               INSTANCE := 'AV-61.02',
               QCMD_OP => "AV-61.02");
END_REGION

REGION Network 23: AV-61.03 w ZSC
   RUNG wire#powerrail
      #"AV-61.03"(AUT_OP := wire#w1, LOCK := #"lock 4", ERR_EXTERN :=, LIOP_SEL := #init, L_AUT := #init, L_REMOTE := #init, L_SIM :=, L_RESET := #reset, MAN_OP :=, SIM_OP :=, FB_OPEN :=, FB_CLOSE :=, L_MON := #init, MON_T :=, MON_T_CLOSE :=, INSTANCE := 'AV-61.03', RESTART :=, VISIBILITY :=, OPdwCmd :=, QdwState =>, QwState =>, QCLOSING =>, QCLOSE =>, QOPENING =>, QOPEN =>, QCMD_OP => "AV-61.03", QMON =>, QMON_ERR =>, QMON_T =>, QMON_T_CLOSE =>, QMAN_AUT =>, QREMOTE =>, QSIM =>, QLOCK =>, QERR =>, QERR_EXT =>, QwAlarm =>)
   END_RUNG
   RUNG wire#powerrail
      Contact( "BFT-61".Out_AV_Inload )
      Contact( "BFT-61".InloadAV_OffTime.Q )
   END_RUNG wire#w1
   // the same network as SCL:
   #"AV-61.03"(LOCK := #"lock 4",   // "Valve"
               LIOP_SEL := #init,
               L_AUT := #init,
               L_REMOTE := #init,
               L_RESET := #reset,
               AUT_OP := "BFT-61".Out_AV_Inload AND "BFT-61".InloadAV_OffTime.Q,
               L_MON := #init,
               INSTANCE := 'AV-61.03',
               QCMD_OP => "AV-61.03");
END_REGION

REGION Network 24: AV-61.04
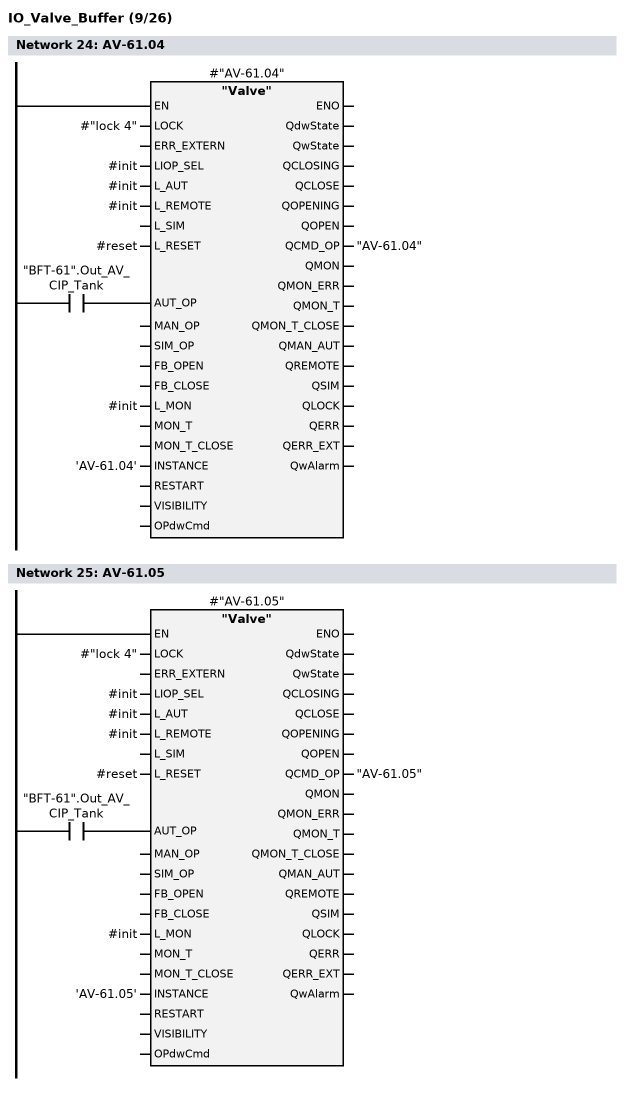
   RUNG wire#powerrail
      #"AV-61.04"(AUT_OP := wire#w1, LOCK := #"lock 4", ERR_EXTERN :=, LIOP_SEL := #init, L_AUT := #init, L_REMOTE := #init, L_SIM :=, L_RESET := #reset, MAN_OP :=, SIM_OP :=, FB_OPEN :=, FB_CLOSE :=, L_MON := #init, MON_T :=, MON_T_CLOSE :=, INSTANCE := 'AV-61.04', RESTART :=, VISIBILITY :=, OPdwCmd :=, QdwState =>, QwState =>, QCLOSING =>, QCLOSE =>, QOPENING =>, QOPEN =>, QCMD_OP => "AV-61.04", QMON =>, QMON_ERR =>, QMON_T =>, QMON_T_CLOSE =>, QMAN_AUT =>, QREMOTE =>, QSIM =>, QLOCK =>, QERR =>, QERR_EXT =>, QwAlarm =>)
   END_RUNG
   RUNG wire#powerrail
      Contact( "BFT-61".Out_AV_CIP_Tank )
   END_RUNG wire#w1
   // the same network as SCL:
   #"AV-61.04"(LOCK := #"lock 4",   // "Valve"
               LIOP_SEL := #init,
               L_AUT := #init,
               L_REMOTE := #init,
               L_RESET := #reset,
               AUT_OP := "BFT-61".Out_AV_CIP_Tank,
               L_MON := #init,
               INSTANCE := 'AV-61.04',
               QCMD_OP => "AV-61.04");
END_REGION

REGION Network 25: AV-61.05
   RUNG wire#powerrail
      #"AV-61.05"(AUT_OP := wire#w1, LOCK := #"lock 4", ERR_EXTERN :=, LIOP_SEL := #init, L_AUT := #init, L_REMOTE := #init, L_SIM :=, L_RESET := #reset, MAN_OP :=, SIM_OP :=, FB_OPEN :=, FB_CLOSE :=, L_MON := #init, MON_T :=, MON_T_CLOSE :=, INSTANCE := 'AV-61.05', RESTART :=, VISIBILITY :=, OPdwCmd :=, QdwState =>, QwState =>, QCLOSING =>, QCLOSE =>, QOPENING =>, QOPEN =>, QCMD_OP => "AV-61.05", QMON =>, QMON_ERR =>, QMON_T =>, QMON_T_CLOSE =>, QMAN_AUT =>, QREMOTE =>, QSIM =>, QLOCK =>, QERR =>, QERR_EXT =>, QwAlarm =>)
   END_RUNG
   RUNG wire#powerrail
      Contact( "BFT-61".Out_AV_CIP_Tank )
   END_RUNG wire#w1
   // the same network as SCL:
   #"AV-61.05"(LOCK := #"lock 4",   // "Valve"
               LIOP_SEL := #init,
               L_AUT := #init,
               L_REMOTE := #init,
               L_RESET := #reset,
               AUT_OP := "BFT-61".Out_AV_CIP_Tank,
               L_MON := #init,
               INSTANCE := 'AV-61.05',
               QCMD_OP => "AV-61.05");
END_REGION

REGION Network 26: AV-61.21
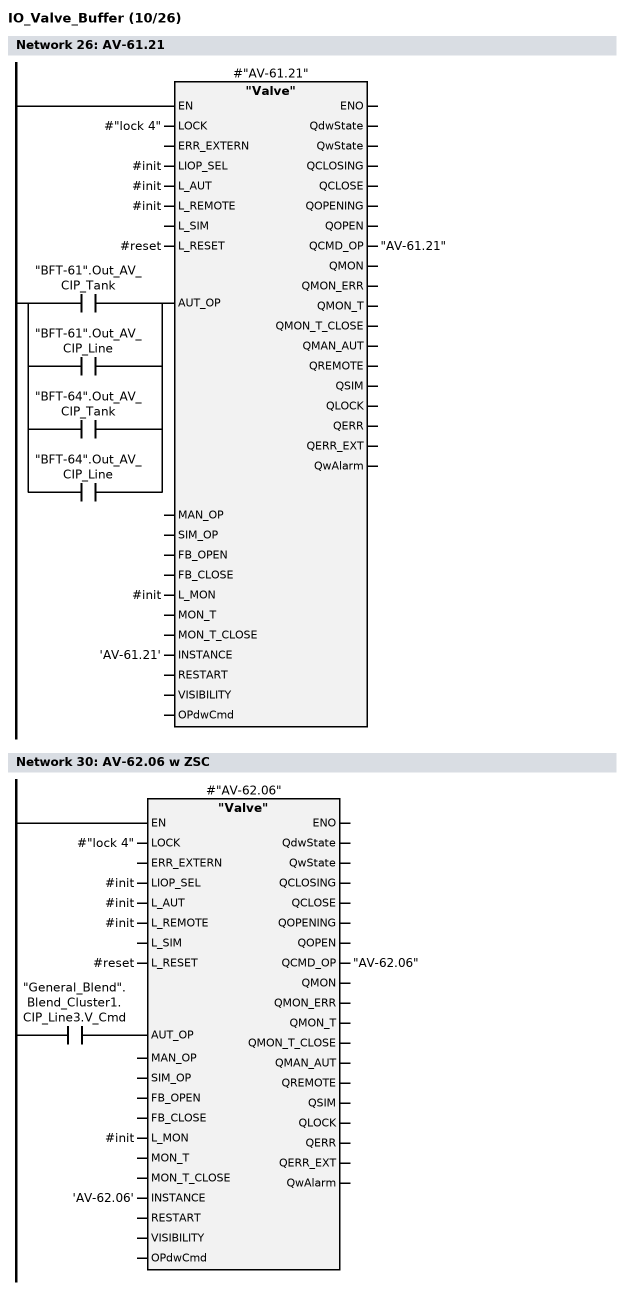
   RUNG wire#powerrail
      #"AV-61.21"(AUT_OP := wire#w1, LOCK := #"lock 4", ERR_EXTERN :=, LIOP_SEL := #init, L_AUT := #init, L_REMOTE := #init, L_SIM :=, L_RESET := #reset, MAN_OP :=, SIM_OP :=, FB_OPEN :=, FB_CLOSE :=, L_MON := #init, MON_T :=, MON_T_CLOSE :=, INSTANCE := 'AV-61.21', RESTART :=, VISIBILITY :=, OPdwCmd :=, QdwState =>, QwState =>, QCLOSING =>, QCLOSE =>, QOPENING =>, QOPEN =>, QCMD_OP => "AV-61.21", QMON =>, QMON_ERR =>, QMON_T =>, QMON_T_CLOSE =>, QMAN_AUT =>, QREMOTE =>, QSIM =>, QLOCK =>, QERR =>, QERR_EXT =>, QwAlarm =>)
   END_RUNG
   RUNG wire#powerrail
      Contact( "BFT-61".Out_AV_CIP_Tank )
   END_RUNG wire#w1
   RUNG wire#powerrail
      Contact( "BFT-61".Out_AV_CIP_Line )
   END_RUNG wire#w1
   RUNG wire#powerrail
      Contact( "BFT-64".Out_AV_CIP_Tank )
   END_RUNG wire#w1
   RUNG wire#powerrail
      Contact( "BFT-64".Out_AV_CIP_Line )
   END_RUNG wire#w1
   // the same network as SCL:
   #"AV-61.21"(LOCK := #"lock 4",   // "Valve"
               LIOP_SEL := #init,
               L_AUT := #init,
               L_REMOTE := #init,
               L_RESET := #reset,
               AUT_OP := "BFT-61".Out_AV_CIP_Tank OR "BFT-61".Out_AV_CIP_Line OR "BFT-64".Out_AV_CIP_Tank OR "BFT-64".Out_AV_CIP_Line,
               L_MON := #init,
               INSTANCE := 'AV-61.21',
               QCMD_OP => "AV-61.21");
END_REGION

REGION Network 28 (SCL): FB OPEN AND CLOSE VALVE T-62
   IF #testing THEN
       // Statement section IF
       #"AV-62.06".FB_OPEN := #"AV-62.06".QCMD_OP;
       #"AV-62.06".FB_CLOSE := NOT #"AV-62.06".QCMD_OP;
   ELSE
       // Statement section ELSE
       #"AV-62.06".FB_OPEN := NOT "ZSC-62.06";
       #"AV-62.06".FB_CLOSE := "ZSC-62.06";
   END_IF;
END_REGION

NETWORK
TITLE = FB MONITORING TIME VALVE T-62
// FB OPEN TIME
      L     T#20s;
      T     #"AV-62.06".MON_T;
// FB CLOSE TIME
      L     T#20s;
      T     #"AV-62.06".MON_T_CLOSE;

REGION Network 30: AV-62.06 w ZSC
   RUNG wire#powerrail
      #"AV-62.06"(AUT_OP := wire#w1, LOCK := #"lock 4", ERR_EXTERN :=, LIOP_SEL := #init, L_AUT := #init, L_REMOTE := #init, L_SIM :=, L_RESET := #reset, MAN_OP :=, SIM_OP :=, FB_OPEN :=, FB_CLOSE :=, L_MON := #init, MON_T :=, MON_T_CLOSE :=, INSTANCE := 'AV-62.06', RESTART :=, VISIBILITY :=, OPdwCmd :=, QdwState =>, QwState =>, QCLOSING =>, QCLOSE =>, QOPENING =>, QOPEN =>, QCMD_OP => "AV-62.06", QMON =>, QMON_ERR =>, QMON_T =>, QMON_T_CLOSE =>, QMAN_AUT =>, QREMOTE =>, QSIM =>, QLOCK =>, QERR =>, QERR_EXT =>, QwAlarm =>)
   END_RUNG
   RUNG wire#powerrail
      Contact( "General_Blend".Blend_Cluster1.CIP_Line3.V_Cmd )
   END_RUNG wire#w1
   // the same network as SCL:
   #"AV-62.06"(LOCK := #"lock 4",   // "Valve"
               LIOP_SEL := #init,
               L_AUT := #init,
               L_REMOTE := #init,
               L_RESET := #reset,
               AUT_OP := "General_Blend".Blend_Cluster1.CIP_Line3.V_Cmd,
               L_MON := #init,
               INSTANCE := 'AV-62.06',
               QCMD_OP => "AV-62.06");
END_REGION

REGION Network 32 (SCL): FB OPEN AND CLOSE VALVE T-64
   IF #testing THEN
       // Statement section IF
       #"AV-64.01".FB_OPEN := #"AV-64.01".QCMD_OP;
       #"AV-64.01".FB_CLOSE := NOT #"AV-64.01".QCMD_OP;
       #"AV-64.02".FB_OPEN := #"AV-64.02".QCMD_OP;
       #"AV-64.02".FB_CLOSE := NOT #"AV-64.02".QCMD_OP;
       #"AV-64.03".FB_OPEN := #"AV-64.03".QCMD_OP;
       #"AV-64.03".FB_CLOSE := NOT #"AV-64.03".QCMD_OP;
       #"AV-64.04".FB_OPEN := #"AV-64.04".QCMD_OP;
       #"AV-64.04".FB_CLOSE := NOT #"AV-64.04".QCMD_OP;
       #"AV-64.05".FB_OPEN := #"AV-64.05".QCMD_OP;
       #"AV-64.05".FB_CLOSE := NOT #"AV-64.05".QCMD_OP;
       #"AV-64.06".FB_OPEN := #"AV-64.06".QCMD_OP;
       #"AV-64.06".FB_CLOSE := NOT #"AV-64.06".QCMD_OP;
   ELSE
       // Statement section ELSE
       #"AV-64.01".FB_OPEN := NOT "ZSC-64.01";
       #"AV-64.01".FB_CLOSE := "ZSC-64.01";
       #"AV-64.02".FB_OPEN := #"AV-64.02".QCMD_OP;
       #"AV-64.02".FB_CLOSE := NOT #"AV-64.02".QCMD_OP;
       #"AV-64.03".FB_OPEN := NOT "ZSC-64.03";
       #"AV-64.03".FB_CLOSE := "ZSC-64.03";
       #"AV-64.04".FB_OPEN := #"AV-64.04".QCMD_OP;
       #"AV-64.04".FB_CLOSE := NOT #"AV-64.04".QCMD_OP;
       #"AV-64.05".FB_OPEN := #"AV-64.05".QCMD_OP;
       #"AV-64.05".FB_CLOSE := NOT #"AV-64.05".QCMD_OP;
       #"AV-64.06".FB_OPEN := NOT "ZSC-64.06";
       #"AV-64.06".FB_CLOSE := "ZSC-64.06";

   END_IF;
END_REGION

NETWORK
TITLE = FB MONITORING TIME VALVE T-64
// FB OPEN TIME
      L     T#20s;
      T     #"AV-64.01".MON_T;
      T     #"AV-64.02".MON_T;
      T     #"AV-64.03".MON_T;
      T     #"AV-64.04".MON_T;
      T     #"AV-64.05".MON_T;
      T     #"AV-64.06".MON_T;
// FB CLOSE TIME
      L     T#20s;
      T     #"AV-64.01".MON_T_CLOSE;
      T     #"AV-64.02".MON_T_CLOSE;
      T     #"AV-64.03".MON_T_CLOSE;
      T     #"AV-64.04".MON_T_CLOSE;
      T     #"AV-64.05".MON_T_CLOSE;
      T     #"AV-64.06".MON_T_CLOSE;

REGION Network 34: AV-64.01 w ZSC
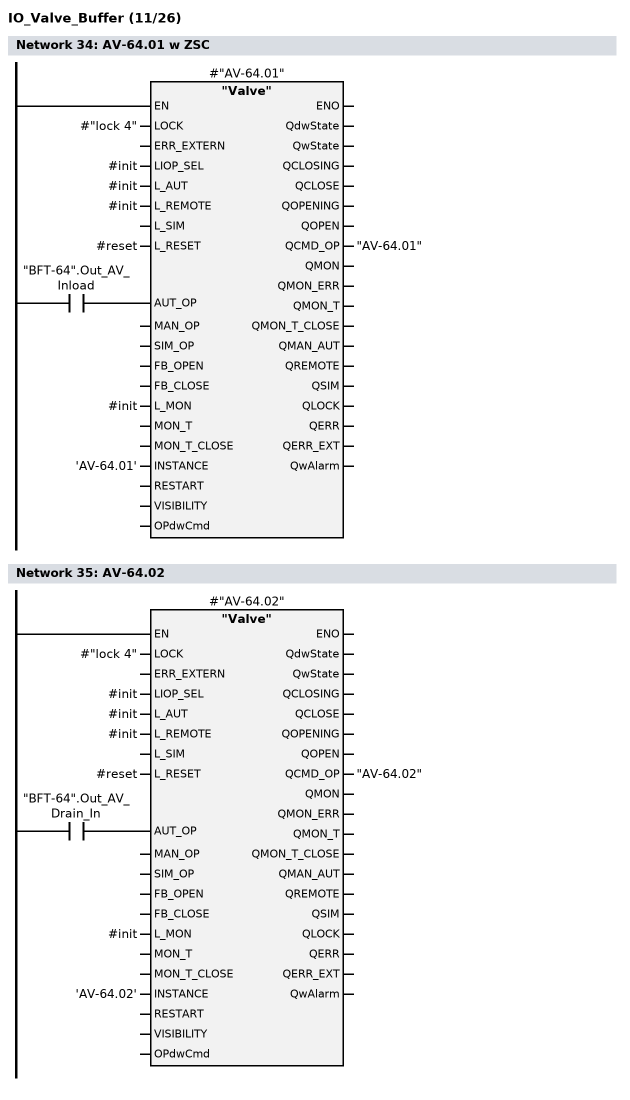
   RUNG wire#powerrail
      #"AV-64.01"(AUT_OP := wire#w1, LOCK := #"lock 4", ERR_EXTERN :=, LIOP_SEL := #init, L_AUT := #init, L_REMOTE := #init, L_SIM :=, L_RESET := #reset, MAN_OP :=, SIM_OP :=, FB_OPEN :=, FB_CLOSE :=, L_MON := #init, MON_T :=, MON_T_CLOSE :=, INSTANCE := 'AV-64.01', RESTART :=, VISIBILITY :=, OPdwCmd :=, QdwState =>, QwState =>, QCLOSING =>, QCLOSE =>, QOPENING =>, QOPEN =>, QCMD_OP => "AV-64.01", QMON =>, QMON_ERR =>, QMON_T =>, QMON_T_CLOSE =>, QMAN_AUT =>, QREMOTE =>, QSIM =>, QLOCK =>, QERR =>, QERR_EXT =>, QwAlarm =>)
   END_RUNG
   RUNG wire#powerrail
      Contact( "BFT-64".Out_AV_Inload )
   END_RUNG wire#w1
   // the same network as SCL:
   #"AV-64.01"(LOCK := #"lock 4",   // "Valve"
               LIOP_SEL := #init,
               L_AUT := #init,
               L_REMOTE := #init,
               L_RESET := #reset,
               AUT_OP := "BFT-64".Out_AV_Inload,
               L_MON := #init,
               INSTANCE := 'AV-64.01',
               QCMD_OP => "AV-64.01");
END_REGION

REGION Network 35: AV-64.02
   RUNG wire#powerrail
      #"AV-64.02"(AUT_OP := wire#w1, LOCK := #"lock 4", ERR_EXTERN :=, LIOP_SEL := #init, L_AUT := #init, L_REMOTE := #init, L_SIM :=, L_RESET := #reset, MAN_OP :=, SIM_OP :=, FB_OPEN :=, FB_CLOSE :=, L_MON := #init, MON_T :=, MON_T_CLOSE :=, INSTANCE := 'AV-64.02', RESTART :=, VISIBILITY :=, OPdwCmd :=, QdwState =>, QwState =>, QCLOSING =>, QCLOSE =>, QOPENING =>, QOPEN =>, QCMD_OP => "AV-64.02", QMON =>, QMON_ERR =>, QMON_T =>, QMON_T_CLOSE =>, QMAN_AUT =>, QREMOTE =>, QSIM =>, QLOCK =>, QERR =>, QERR_EXT =>, QwAlarm =>)
   END_RUNG
   RUNG wire#powerrail
      Contact( "BFT-64".Out_AV_Drain_In )
   END_RUNG wire#w1
   // the same network as SCL:
   #"AV-64.02"(LOCK := #"lock 4",   // "Valve"
               LIOP_SEL := #init,
               L_AUT := #init,
               L_REMOTE := #init,
               L_RESET := #reset,
               AUT_OP := "BFT-64".Out_AV_Drain_In,
               L_MON := #init,
               INSTANCE := 'AV-64.02',
               QCMD_OP => "AV-64.02");
END_REGION

REGION Network 36: AV-64.03 w ZSC
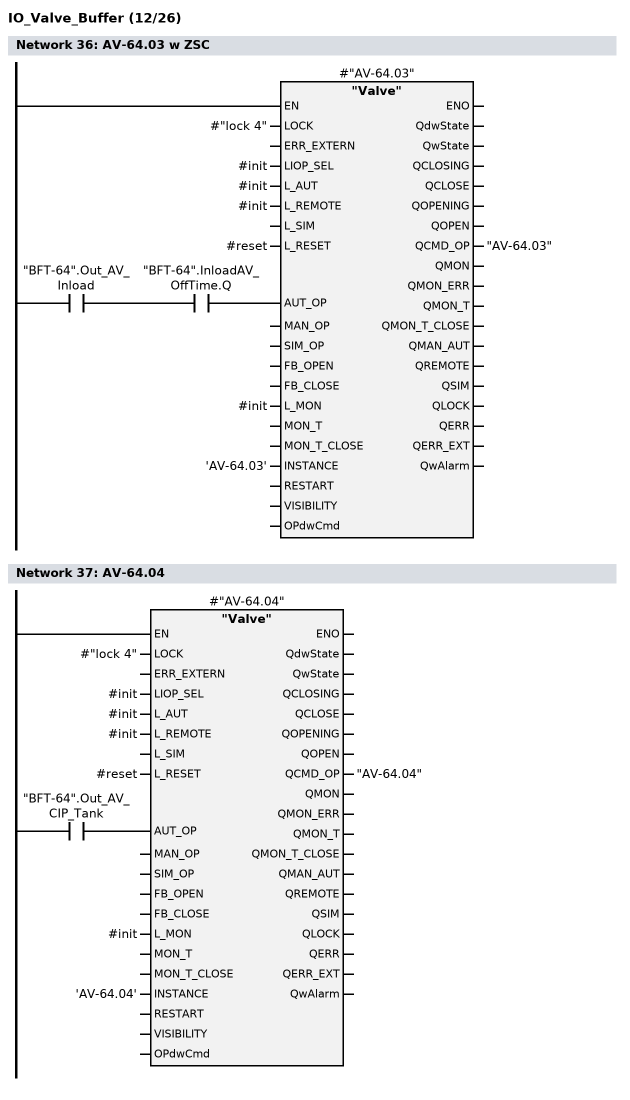
   RUNG wire#powerrail
      #"AV-64.03"(AUT_OP := wire#w1, LOCK := #"lock 4", ERR_EXTERN :=, LIOP_SEL := #init, L_AUT := #init, L_REMOTE := #init, L_SIM :=, L_RESET := #reset, MAN_OP :=, SIM_OP :=, FB_OPEN :=, FB_CLOSE :=, L_MON := #init, MON_T :=, MON_T_CLOSE :=, INSTANCE := 'AV-64.03', RESTART :=, VISIBILITY :=, OPdwCmd :=, QdwState =>, QwState =>, QCLOSING =>, QCLOSE =>, QOPENING =>, QOPEN =>, QCMD_OP => "AV-64.03", QMON =>, QMON_ERR =>, QMON_T =>, QMON_T_CLOSE =>, QMAN_AUT =>, QREMOTE =>, QSIM =>, QLOCK =>, QERR =>, QERR_EXT =>, QwAlarm =>)
   END_RUNG
   RUNG wire#powerrail
      Contact( "BFT-64".Out_AV_Inload )
      Contact( "BFT-64".InloadAV_OffTime.Q )
   END_RUNG wire#w1
   // the same network as SCL:
   #"AV-64.03"(LOCK := #"lock 4",   // "Valve"
               LIOP_SEL := #init,
               L_AUT := #init,
               L_REMOTE := #init,
               L_RESET := #reset,
               AUT_OP := "BFT-64".Out_AV_Inload AND "BFT-64".InloadAV_OffTime.Q,
               L_MON := #init,
               INSTANCE := 'AV-64.03',
               QCMD_OP => "AV-64.03");
END_REGION

REGION Network 37: AV-64.04
   RUNG wire#powerrail
      #"AV-64.04"(AUT_OP := wire#w1, LOCK := #"lock 4", ERR_EXTERN :=, LIOP_SEL := #init, L_AUT := #init, L_REMOTE := #init, L_SIM :=, L_RESET := #reset, MAN_OP :=, SIM_OP :=, FB_OPEN :=, FB_CLOSE :=, L_MON := #init, MON_T :=, MON_T_CLOSE :=, INSTANCE := 'AV-64.04', RESTART :=, VISIBILITY :=, OPdwCmd :=, QdwState =>, QwState =>, QCLOSING =>, QCLOSE =>, QOPENING =>, QOPEN =>, QCMD_OP => "AV-64.04", QMON =>, QMON_ERR =>, QMON_T =>, QMON_T_CLOSE =>, QMAN_AUT =>, QREMOTE =>, QSIM =>, QLOCK =>, QERR =>, QERR_EXT =>, QwAlarm =>)
   END_RUNG
   RUNG wire#powerrail
      Contact( "BFT-64".Out_AV_CIP_Tank )
   END_RUNG wire#w1
   // the same network as SCL:
   #"AV-64.04"(LOCK := #"lock 4",   // "Valve"
               LIOP_SEL := #init,
               L_AUT := #init,
               L_REMOTE := #init,
               L_RESET := #reset,
               AUT_OP := "BFT-64".Out_AV_CIP_Tank,
               L_MON := #init,
               INSTANCE := 'AV-64.04',
               QCMD_OP => "AV-64.04");
END_REGION

REGION Network 38: AV-64.05
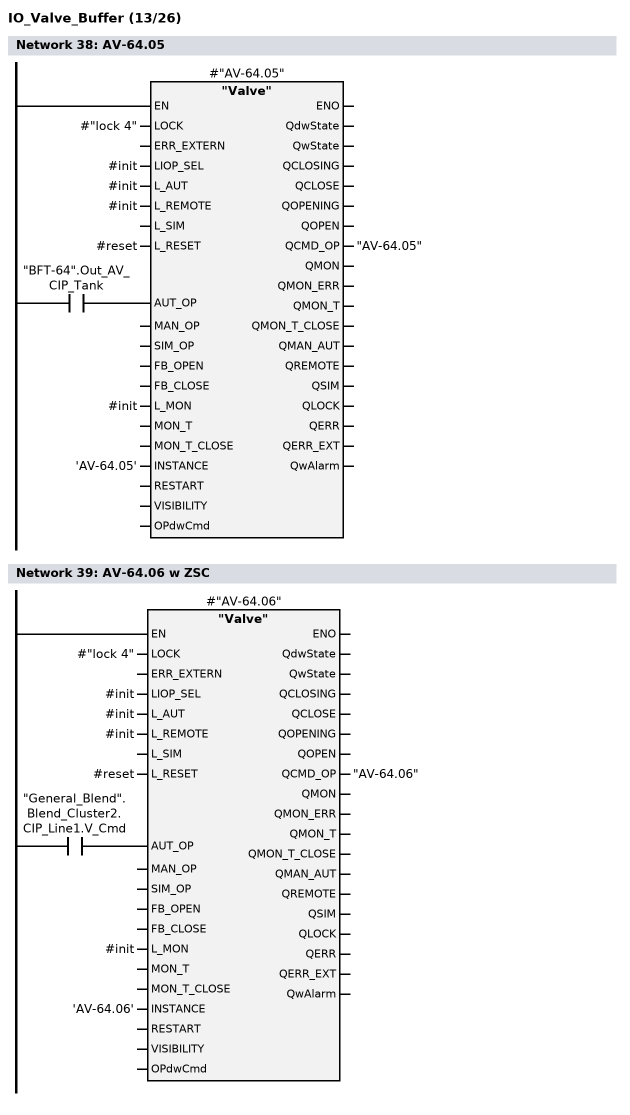
   RUNG wire#powerrail
      #"AV-64.05"(AUT_OP := wire#w1, LOCK := #"lock 4", ERR_EXTERN :=, LIOP_SEL := #init, L_AUT := #init, L_REMOTE := #init, L_SIM :=, L_RESET := #reset, MAN_OP :=, SIM_OP :=, FB_OPEN :=, FB_CLOSE :=, L_MON := #init, MON_T :=, MON_T_CLOSE :=, INSTANCE := 'AV-64.05', RESTART :=, VISIBILITY :=, OPdwCmd :=, QdwState =>, QwState =>, QCLOSING =>, QCLOSE =>, QOPENING =>, QOPEN =>, QCMD_OP => "AV-64.05", QMON =>, QMON_ERR =>, QMON_T =>, QMON_T_CLOSE =>, QMAN_AUT =>, QREMOTE =>, QSIM =>, QLOCK =>, QERR =>, QERR_EXT =>, QwAlarm =>)
   END_RUNG
   RUNG wire#powerrail
      Contact( "BFT-64".Out_AV_CIP_Tank )
   END_RUNG wire#w1
   // the same network as SCL:
   #"AV-64.05"(LOCK := #"lock 4",   // "Valve"
               LIOP_SEL := #init,
               L_AUT := #init,
               L_REMOTE := #init,
               L_RESET := #reset,
               AUT_OP := "BFT-64".Out_AV_CIP_Tank,
               L_MON := #init,
               INSTANCE := 'AV-64.05',
               QCMD_OP => "AV-64.05");
END_REGION

REGION Network 39: AV-64.06 w ZSC
   RUNG wire#powerrail
      #"AV-64.06"(AUT_OP := wire#w1, LOCK := #"lock 4", ERR_EXTERN :=, LIOP_SEL := #init, L_AUT := #init, L_REMOTE := #init, L_SIM :=, L_RESET := #reset, MAN_OP :=, SIM_OP :=, FB_OPEN :=, FB_CLOSE :=, L_MON := #init, MON_T :=, MON_T_CLOSE :=, INSTANCE := 'AV-64.06', RESTART :=, VISIBILITY :=, OPdwCmd :=, QdwState =>, QwState =>, QCLOSING =>, QCLOSE =>, QOPENING =>, QOPEN =>, QCMD_OP => "AV-64.06", QMON =>, QMON_ERR =>, QMON_T =>, QMON_T_CLOSE =>, QMAN_AUT =>, QREMOTE =>, QSIM =>, QLOCK =>, QERR =>, QERR_EXT =>, QwAlarm =>)
   END_RUNG
   RUNG wire#powerrail
      Contact( "General_Blend".Blend_Cluster2.CIP_Line1.V_Cmd )
   END_RUNG wire#w1
   // the same network as SCL:
   #"AV-64.06"(LOCK := #"lock 4",   // "Valve"
               LIOP_SEL := #init,
               L_AUT := #init,
               L_REMOTE := #init,
               L_RESET := #reset,
               AUT_OP := "General_Blend".Blend_Cluster2.CIP_Line1.V_Cmd,
               L_MON := #init,
               INSTANCE := 'AV-64.06',
               QCMD_OP => "AV-64.06");
END_REGION

REGION Network 41 (SCL): FB OPEN AND CLOSE VALVE T-65
   IF #testing THEN
       // Statement section IF
       #"AV-65.01".FB_OPEN := #"AV-65.01".QCMD_OP;
       #"AV-65.01".FB_CLOSE := NOT #"AV-65.01".QCMD_OP;
       #"AV-65.02".FB_OPEN := #"AV-65.02".QCMD_OP;
       #"AV-65.02".FB_CLOSE := NOT #"AV-65.02".QCMD_OP;
       #"AV-65.03".FB_OPEN := #"AV-65.03".QCMD_OP;
       #"AV-65.03".FB_CLOSE := NOT #"AV-65.03".QCMD_OP;
       #"AV-65.04".FB_OPEN := #"AV-65.04".QCMD_OP;
       #"AV-65.04".FB_CLOSE := NOT #"AV-65.04".QCMD_OP;
       #"AV-65.05".FB_OPEN := #"AV-65.05".QCMD_OP;
       #"AV-65.05".FB_CLOSE := NOT #"AV-65.05".QCMD_OP;
       #"AV-65.21".FB_OPEN := #"AV-65.21".QCMD_OP;
       #"AV-65.21".FB_CLOSE := NOT #"AV-65.21".QCMD_OP;
   ELSE
       // Statement section ELSE
       #"AV-65.01".FB_OPEN := NOT "ZSC-65.01";
       #"AV-65.01".FB_CLOSE := "ZSC-65.01";
       #"AV-65.02".FB_OPEN := #"AV-65.02".QCMD_OP;
       #"AV-65.02".FB_CLOSE := NOT #"AV-65.02".QCMD_OP;
       #"AV-65.03".FB_OPEN := NOT "ZSC-65.03";
       #"AV-65.03".FB_CLOSE := "ZSC-65.03";
       #"AV-65.04".FB_OPEN := #"AV-65.04".QCMD_OP;
       #"AV-65.04".FB_CLOSE := NOT #"AV-65.04".QCMD_OP;
       #"AV-65.05".FB_OPEN := #"AV-65.05".QCMD_OP;
       #"AV-65.05".FB_CLOSE := NOT #"AV-65.05".QCMD_OP;
       #"AV-65.21".FB_OPEN := #"AV-65.21".QCMD_OP;
       #"AV-65.21".FB_CLOSE := NOT #"AV-65.21".QCMD_OP;
   END_IF;
END_REGION

NETWORK
TITLE = FB MONITORING TIME VALVE T-65
// FB OPEN TIME
      L     T#20s;
      T     #"AV-65.01".MON_T;
      T     #"AV-65.02".MON_T;
      T     #"AV-65.03".MON_T;
      T     #"AV-65.04".MON_T;
      T     #"AV-65.05".MON_T;
      T     #"AV-65.21".MON_T;
// FB CLOSE TIME
      L     T#20s;
      T     #"AV-65.01".MON_T_CLOSE;
      T     #"AV-65.02".MON_T_CLOSE;
      T     #"AV-65.03".MON_T_CLOSE;
      T     #"AV-65.04".MON_T_CLOSE;
      T     #"AV-65.05".MON_T_CLOSE;
      T     #"AV-65.21".MON_T_CLOSE;

REGION Network 43: AV-65.01 w ZSC
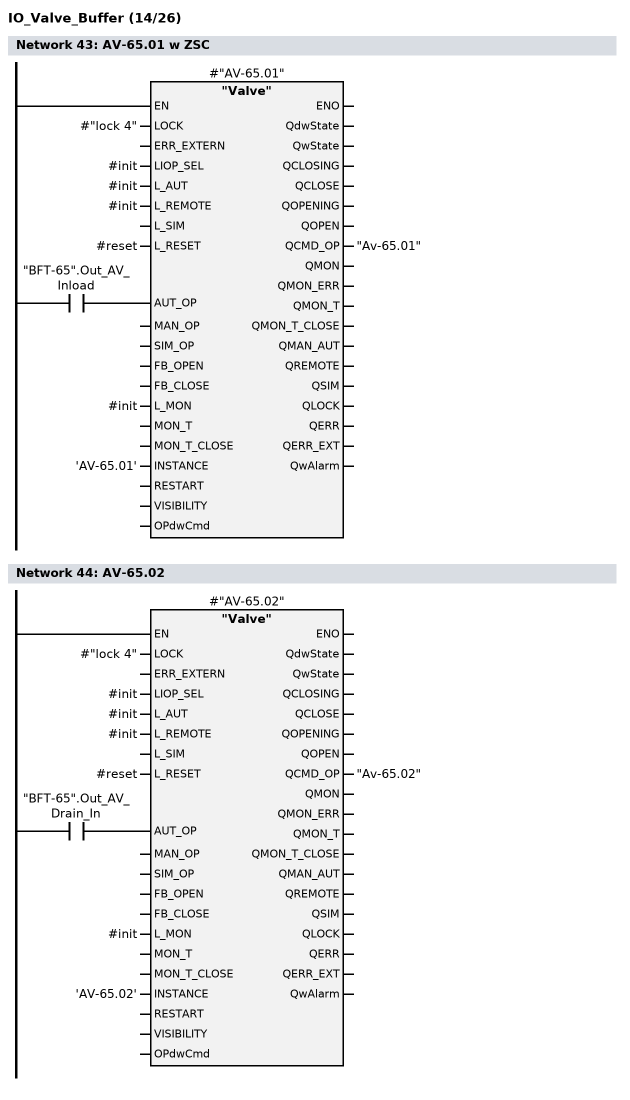
   RUNG wire#powerrail
      #"AV-65.01"(AUT_OP := wire#w1, LOCK := #"lock 4", ERR_EXTERN :=, LIOP_SEL := #init, L_AUT := #init, L_REMOTE := #init, L_SIM :=, L_RESET := #reset, MAN_OP :=, SIM_OP :=, FB_OPEN :=, FB_CLOSE :=, L_MON := #init, MON_T :=, MON_T_CLOSE :=, INSTANCE := 'AV-65.01', RESTART :=, VISIBILITY :=, OPdwCmd :=, QdwState =>, QwState =>, QCLOSING =>, QCLOSE =>, QOPENING =>, QOPEN =>, QCMD_OP => "Av-65.01", QMON =>, QMON_ERR =>, QMON_T =>, QMON_T_CLOSE =>, QMAN_AUT =>, QREMOTE =>, QSIM =>, QLOCK =>, QERR =>, QERR_EXT =>, QwAlarm =>)
   END_RUNG
   RUNG wire#powerrail
      Contact( "BFT-65".Out_AV_Inload )
   END_RUNG wire#w1
   // the same network as SCL:
   #"AV-65.01"(LOCK := #"lock 4",   // "Valve"
               LIOP_SEL := #init,
               L_AUT := #init,
               L_REMOTE := #init,
               L_RESET := #reset,
               AUT_OP := "BFT-65".Out_AV_Inload,
               L_MON := #init,
               INSTANCE := 'AV-65.01',
               QCMD_OP => "Av-65.01");
END_REGION

REGION Network 44: AV-65.02
   RUNG wire#powerrail
      #"AV-65.02"(AUT_OP := wire#w1, LOCK := #"lock 4", ERR_EXTERN :=, LIOP_SEL := #init, L_AUT := #init, L_REMOTE := #init, L_SIM :=, L_RESET := #reset, MAN_OP :=, SIM_OP :=, FB_OPEN :=, FB_CLOSE :=, L_MON := #init, MON_T :=, MON_T_CLOSE :=, INSTANCE := 'AV-65.02', RESTART :=, VISIBILITY :=, OPdwCmd :=, QdwState =>, QwState =>, QCLOSING =>, QCLOSE =>, QOPENING =>, QOPEN =>, QCMD_OP => "Av-65.02", QMON =>, QMON_ERR =>, QMON_T =>, QMON_T_CLOSE =>, QMAN_AUT =>, QREMOTE =>, QSIM =>, QLOCK =>, QERR =>, QERR_EXT =>, QwAlarm =>)
   END_RUNG
   RUNG wire#powerrail
      Contact( "BFT-65".Out_AV_Drain_In )
   END_RUNG wire#w1
   // the same network as SCL:
   #"AV-65.02"(LOCK := #"lock 4",   // "Valve"
               LIOP_SEL := #init,
               L_AUT := #init,
               L_REMOTE := #init,
               L_RESET := #reset,
               AUT_OP := "BFT-65".Out_AV_Drain_In,
               L_MON := #init,
               INSTANCE := 'AV-65.02',
               QCMD_OP => "Av-65.02");
END_REGION

REGION Network 45: AV-65.03 w ZSC
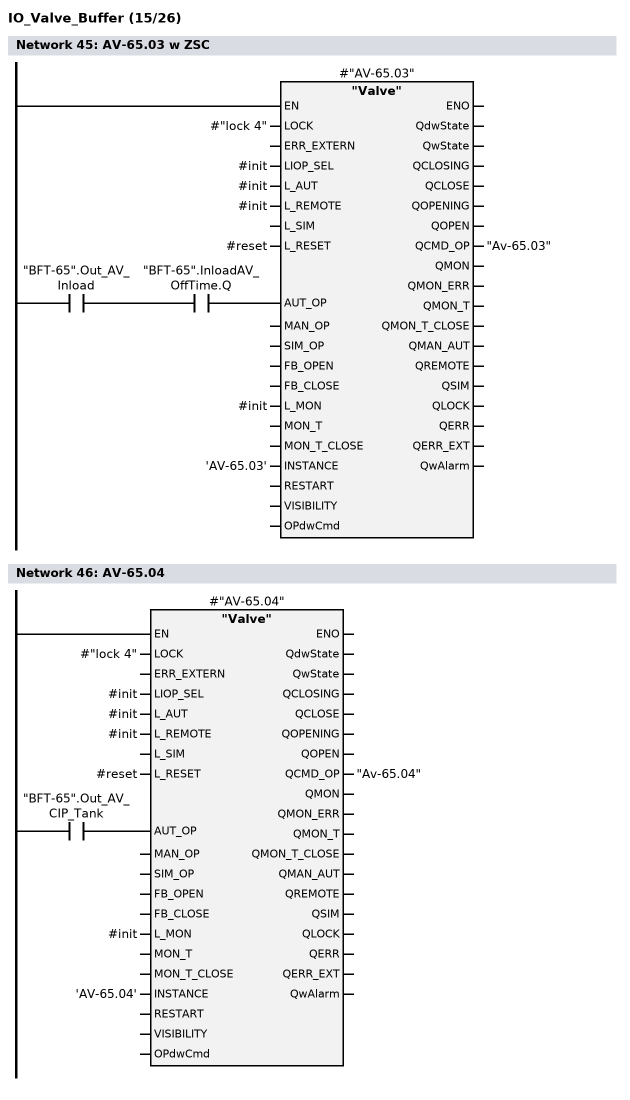
   RUNG wire#powerrail
      #"AV-65.03"(AUT_OP := wire#w1, LOCK := #"lock 4", ERR_EXTERN :=, LIOP_SEL := #init, L_AUT := #init, L_REMOTE := #init, L_SIM :=, L_RESET := #reset, MAN_OP :=, SIM_OP :=, FB_OPEN :=, FB_CLOSE :=, L_MON := #init, MON_T :=, MON_T_CLOSE :=, INSTANCE := 'AV-65.03', RESTART :=, VISIBILITY :=, OPdwCmd :=, QdwState =>, QwState =>, QCLOSING =>, QCLOSE =>, QOPENING =>, QOPEN =>, QCMD_OP => "Av-65.03", QMON =>, QMON_ERR =>, QMON_T =>, QMON_T_CLOSE =>, QMAN_AUT =>, QREMOTE =>, QSIM =>, QLOCK =>, QERR =>, QERR_EXT =>, QwAlarm =>)
   END_RUNG
   RUNG wire#powerrail
      Contact( "BFT-65".Out_AV_Inload )
      Contact( "BFT-65".InloadAV_OffTime.Q )
   END_RUNG wire#w1
   // the same network as SCL:
   #"AV-65.03"(LOCK := #"lock 4",   // "Valve"
               LIOP_SEL := #init,
               L_AUT := #init,
               L_REMOTE := #init,
               L_RESET := #reset,
               AUT_OP := "BFT-65".Out_AV_Inload AND "BFT-65".InloadAV_OffTime.Q,
               L_MON := #init,
               INSTANCE := 'AV-65.03',
               QCMD_OP => "Av-65.03");
END_REGION

REGION Network 46: AV-65.04
   RUNG wire#powerrail
      #"AV-65.04"(AUT_OP := wire#w1, LOCK := #"lock 4", ERR_EXTERN :=, LIOP_SEL := #init, L_AUT := #init, L_REMOTE := #init, L_SIM :=, L_RESET := #reset, MAN_OP :=, SIM_OP :=, FB_OPEN :=, FB_CLOSE :=, L_MON := #init, MON_T :=, MON_T_CLOSE :=, INSTANCE := 'AV-65.04', RESTART :=, VISIBILITY :=, OPdwCmd :=, QdwState =>, QwState =>, QCLOSING =>, QCLOSE =>, QOPENING =>, QOPEN =>, QCMD_OP => "Av-65.04", QMON =>, QMON_ERR =>, QMON_T =>, QMON_T_CLOSE =>, QMAN_AUT =>, QREMOTE =>, QSIM =>, QLOCK =>, QERR =>, QERR_EXT =>, QwAlarm =>)
   END_RUNG
   RUNG wire#powerrail
      Contact( "BFT-65".Out_AV_CIP_Tank )
   END_RUNG wire#w1
   // the same network as SCL:
   #"AV-65.04"(LOCK := #"lock 4",   // "Valve"
               LIOP_SEL := #init,
               L_AUT := #init,
               L_REMOTE := #init,
               L_RESET := #reset,
               AUT_OP := "BFT-65".Out_AV_CIP_Tank,
               L_MON := #init,
               INSTANCE := 'AV-65.04',
               QCMD_OP => "Av-65.04");
END_REGION

REGION Network 47: AV-65.05
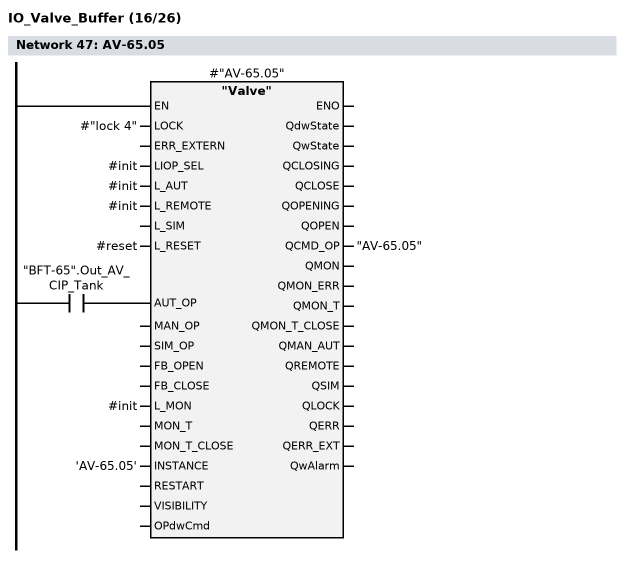
   RUNG wire#powerrail
      #"AV-65.05"(AUT_OP := wire#w1, LOCK := #"lock 4", ERR_EXTERN :=, LIOP_SEL := #init, L_AUT := #init, L_REMOTE := #init, L_SIM :=, L_RESET := #reset, MAN_OP :=, SIM_OP :=, FB_OPEN :=, FB_CLOSE :=, L_MON := #init, MON_T :=, MON_T_CLOSE :=, INSTANCE := 'AV-65.05', RESTART :=, VISIBILITY :=, OPdwCmd :=, QdwState =>, QwState =>, QCLOSING =>, QCLOSE =>, QOPENING =>, QOPEN =>, QCMD_OP => "AV-65.05", QMON =>, QMON_ERR =>, QMON_T =>, QMON_T_CLOSE =>, QMAN_AUT =>, QREMOTE =>, QSIM =>, QLOCK =>, QERR =>, QERR_EXT =>, QwAlarm =>)
   END_RUNG
   RUNG wire#powerrail
      Contact( "BFT-65".Out_AV_CIP_Tank )
   END_RUNG wire#w1
   // the same network as SCL:
   #"AV-65.05"(LOCK := #"lock 4",   // "Valve"
               LIOP_SEL := #init,
               L_AUT := #init,
               L_REMOTE := #init,
               L_RESET := #reset,
               AUT_OP := "BFT-65".Out_AV_CIP_Tank,
               L_MON := #init,
               INSTANCE := 'AV-65.05',
               QCMD_OP => "AV-65.05");
END_REGION

REGION Network 48: AV-65.21
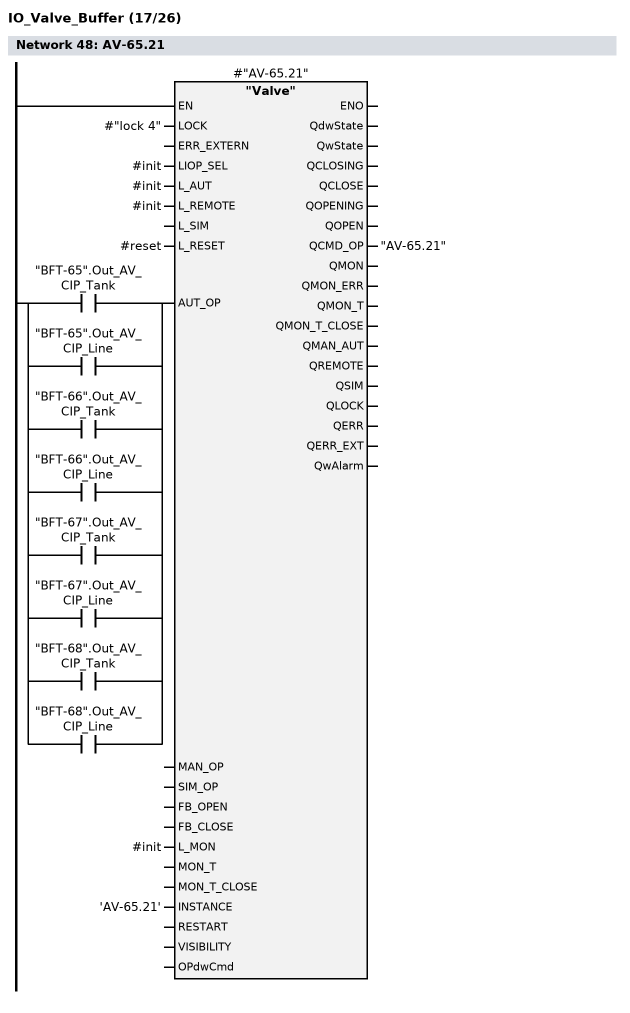
   RUNG wire#powerrail
      #"AV-65.21"(AUT_OP := wire#w1, LOCK := #"lock 4", ERR_EXTERN :=, LIOP_SEL := #init, L_AUT := #init, L_REMOTE := #init, L_SIM :=, L_RESET := #reset, MAN_OP :=, SIM_OP :=, FB_OPEN :=, FB_CLOSE :=, L_MON := #init, MON_T :=, MON_T_CLOSE :=, INSTANCE := 'AV-65.21', RESTART :=, VISIBILITY :=, OPdwCmd :=, QdwState =>, QwState =>, QCLOSING =>, QCLOSE =>, QOPENING =>, QOPEN =>, QCMD_OP => "AV-65.21", QMON =>, QMON_ERR =>, QMON_T =>, QMON_T_CLOSE =>, QMAN_AUT =>, QREMOTE =>, QSIM =>, QLOCK =>, QERR =>, QERR_EXT =>, QwAlarm =>)
   END_RUNG
   RUNG wire#powerrail
      Contact( "BFT-65".Out_AV_CIP_Tank )
   END_RUNG wire#w1
   RUNG wire#powerrail
      Contact( "BFT-65".Out_AV_CIP_Line )
   END_RUNG wire#w1
   RUNG wire#powerrail
      Contact( "BFT-66".Out_AV_CIP_Tank )
   END_RUNG wire#w1
   RUNG wire#powerrail
      Contact( "BFT-66".Out_AV_CIP_Line )
   END_RUNG wire#w1
   RUNG wire#powerrail
      Contact( "BFT-67".Out_AV_CIP_Tank )
   END_RUNG wire#w1
   RUNG wire#powerrail
      Contact( "BFT-67".Out_AV_CIP_Line )
   END_RUNG wire#w1
   RUNG wire#powerrail
      Contact( "BFT-68".Out_AV_CIP_Tank )
   END_RUNG wire#w1
   RUNG wire#powerrail
      Contact( "BFT-68".Out_AV_CIP_Line )
   END_RUNG wire#w1
   // the same network as SCL:
   #"AV-65.21"(LOCK := #"lock 4",   // "Valve"
               LIOP_SEL := #init,
               L_AUT := #init,
               L_REMOTE := #init,
               L_RESET := #reset,
               AUT_OP := "BFT-65".Out_AV_CIP_Tank OR "BFT-65".Out_AV_CIP_Line OR "BFT-66".Out_AV_CIP_Tank OR "BFT-66".Out_AV_CIP_Line OR "BFT-67".Out_AV_CIP_Tank OR "BFT-67".Out_AV_CIP_Line OR "BFT-68".Out_AV_CIP_Tank OR "BFT-68".Out_AV_CIP_Line,
               L_MON := #init,
               INSTANCE := 'AV-65.21',
               QCMD_OP => "AV-65.21");
END_REGION

REGION Network 50 (SCL): FB OPEN AND CLOSE VALVE T-66
   IF #testing THEN
       // Statement section IF
       #"AV-66.01".FB_OPEN := #"AV-66.01".QCMD_OP;
       #"AV-66.01".FB_CLOSE := NOT #"AV-66.01".QCMD_OP;
       #"AV-66.02".FB_OPEN := #"AV-66.02".QCMD_OP;
       #"AV-66.02".FB_CLOSE := NOT #"AV-66.02".QCMD_OP;
       #"AV-66.03".FB_OPEN := #"AV-66.03".QCMD_OP;
       #"AV-66.03".FB_CLOSE := NOT #"AV-66.03".QCMD_OP;
       #"AV-66.04".FB_OPEN := #"AV-66.04".QCMD_OP;
       #"AV-66.04".FB_CLOSE := NOT #"AV-66.04".QCMD_OP;
       #"AV-66.05".FB_OPEN := #"AV-66.05".QCMD_OP;
       #"AV-66.05".FB_CLOSE := NOT #"AV-66.05".QCMD_OP;
       #"AV-66.06".FB_OPEN := #"AV-66.06".QCMD_OP;
       #"AV-66.06".FB_CLOSE := NOT #"AV-66.06".QCMD_OP;
   ELSE
       // Statement section ELSE
       #"AV-66.01".FB_OPEN := NOT "ZSC-66.01";
       #"AV-66.01".FB_CLOSE := "ZSC-66.01";
       #"AV-66.02".FB_OPEN := #"AV-66.02".QCMD_OP;
       #"AV-66.02".FB_CLOSE := NOT #"AV-66.02".QCMD_OP;
       #"AV-66.03".FB_OPEN := NOT "ZSC-66.03";
       #"AV-66.03".FB_CLOSE := "ZSC-66.03";
       #"AV-66.04".FB_OPEN := #"AV-66.04".QCMD_OP;
       #"AV-66.04".FB_CLOSE := NOT #"AV-66.04".QCMD_OP;
       #"AV-66.05".FB_OPEN := #"AV-66.05".QCMD_OP;
       #"AV-66.05".FB_CLOSE := NOT #"AV-66.05".QCMD_OP;
       #"AV-66.06".FB_OPEN := NOT "ZSC-66.06";
       #"AV-66.06".FB_CLOSE := "ZSC-66.06";
   END_IF;
END_REGION

NETWORK
TITLE = FB MONITORING TIME VALVE T-66
// FB OPEN TIME
      L     T#20s;
      T     #"AV-66.01".MON_T;
      T     #"AV-66.02".MON_T;
      T     #"AV-66.03".MON_T;
      T     #"AV-66.04".MON_T;
      T     #"AV-66.05".MON_T;
      T     #"AV-66.06".MON_T;
// FB CLOSE TIME
      L     T#20s;
      T     #"AV-66.01".MON_T_CLOSE;
      T     #"AV-66.02".MON_T_CLOSE;
      T     #"AV-66.03".MON_T_CLOSE;
      T     #"AV-66.04".MON_T_CLOSE;
      T     #"AV-66.05".MON_T_CLOSE;
      T     #"AV-66.06".MON_T_CLOSE;

REGION Network 52: AV-66.01 w ZSC
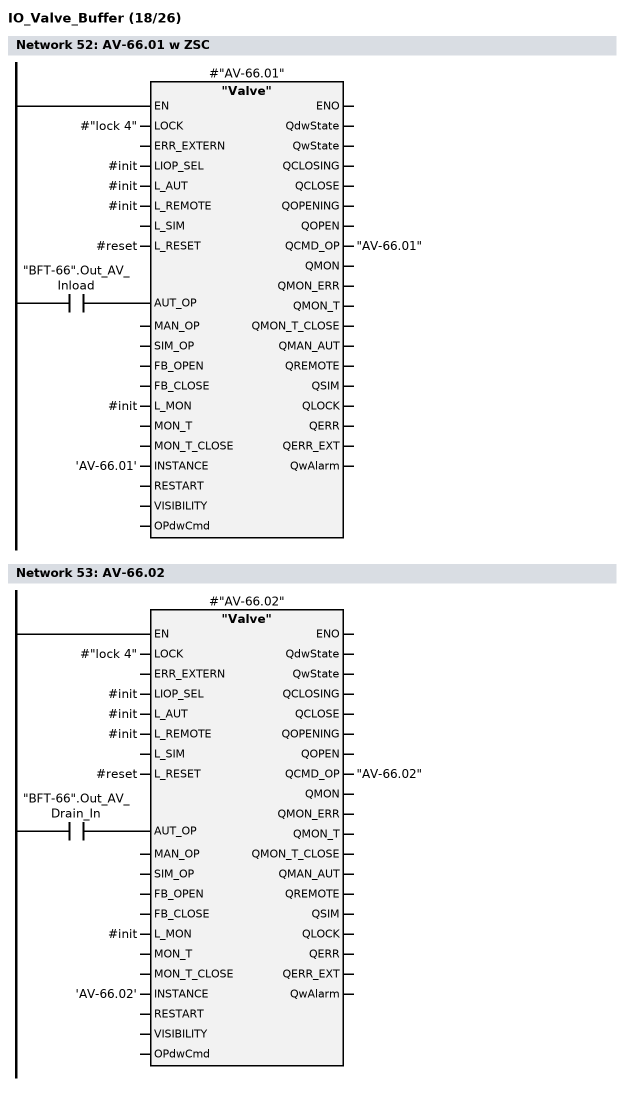
   RUNG wire#powerrail
      #"AV-66.01"(AUT_OP := wire#w1, LOCK := #"lock 4", ERR_EXTERN :=, LIOP_SEL := #init, L_AUT := #init, L_REMOTE := #init, L_SIM :=, L_RESET := #reset, MAN_OP :=, SIM_OP :=, FB_OPEN :=, FB_CLOSE :=, L_MON := #init, MON_T :=, MON_T_CLOSE :=, INSTANCE := 'AV-66.01', RESTART :=, VISIBILITY :=, OPdwCmd :=, QdwState =>, QwState =>, QCLOSING =>, QCLOSE =>, QOPENING =>, QOPEN =>, QCMD_OP => "AV-66.01", QMON =>, QMON_ERR =>, QMON_T =>, QMON_T_CLOSE =>, QMAN_AUT =>, QREMOTE =>, QSIM =>, QLOCK =>, QERR =>, QERR_EXT =>, QwAlarm =>)
   END_RUNG
   RUNG wire#powerrail
      Contact( "BFT-66".Out_AV_Inload )
   END_RUNG wire#w1
   // the same network as SCL:
   #"AV-66.01"(LOCK := #"lock 4",   // "Valve"
               LIOP_SEL := #init,
               L_AUT := #init,
               L_REMOTE := #init,
               L_RESET := #reset,
               AUT_OP := "BFT-66".Out_AV_Inload,
               L_MON := #init,
               INSTANCE := 'AV-66.01',
               QCMD_OP => "AV-66.01");
END_REGION

REGION Network 53: AV-66.02
   RUNG wire#powerrail
      #"AV-66.02"(AUT_OP := wire#w1, LOCK := #"lock 4", ERR_EXTERN :=, LIOP_SEL := #init, L_AUT := #init, L_REMOTE := #init, L_SIM :=, L_RESET := #reset, MAN_OP :=, SIM_OP :=, FB_OPEN :=, FB_CLOSE :=, L_MON := #init, MON_T :=, MON_T_CLOSE :=, INSTANCE := 'AV-66.02', RESTART :=, VISIBILITY :=, OPdwCmd :=, QdwState =>, QwState =>, QCLOSING =>, QCLOSE =>, QOPENING =>, QOPEN =>, QCMD_OP => "AV-66.02", QMON =>, QMON_ERR =>, QMON_T =>, QMON_T_CLOSE =>, QMAN_AUT =>, QREMOTE =>, QSIM =>, QLOCK =>, QERR =>, QERR_EXT =>, QwAlarm =>)
   END_RUNG
   RUNG wire#powerrail
      Contact( "BFT-66".Out_AV_Drain_In )
   END_RUNG wire#w1
   // the same network as SCL:
   #"AV-66.02"(LOCK := #"lock 4",   // "Valve"
               LIOP_SEL := #init,
               L_AUT := #init,
               L_REMOTE := #init,
               L_RESET := #reset,
               AUT_OP := "BFT-66".Out_AV_Drain_In,
               L_MON := #init,
               INSTANCE := 'AV-66.02',
               QCMD_OP => "AV-66.02");
END_REGION

REGION Network 54: AV-66.03 w ZSC
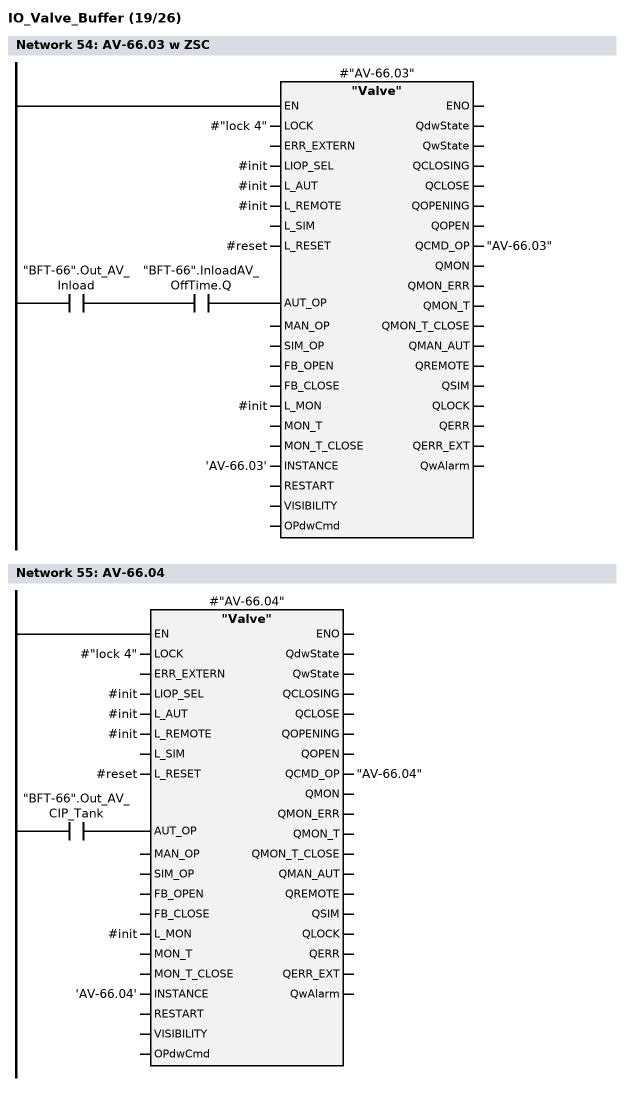
   RUNG wire#powerrail
      #"AV-66.03"(AUT_OP := wire#w1, LOCK := #"lock 4", ERR_EXTERN :=, LIOP_SEL := #init, L_AUT := #init, L_REMOTE := #init, L_SIM :=, L_RESET := #reset, MAN_OP :=, SIM_OP :=, FB_OPEN :=, FB_CLOSE :=, L_MON := #init, MON_T :=, MON_T_CLOSE :=, INSTANCE := 'AV-66.03', RESTART :=, VISIBILITY :=, OPdwCmd :=, QdwState =>, QwState =>, QCLOSING =>, QCLOSE =>, QOPENING =>, QOPEN =>, QCMD_OP => "AV-66.03", QMON =>, QMON_ERR =>, QMON_T =>, QMON_T_CLOSE =>, QMAN_AUT =>, QREMOTE =>, QSIM =>, QLOCK =>, QERR =>, QERR_EXT =>, QwAlarm =>)
   END_RUNG
   RUNG wire#powerrail
      Contact( "BFT-66".Out_AV_Inload )
      Contact( "BFT-66".InloadAV_OffTime.Q )
   END_RUNG wire#w1
   // the same network as SCL:
   #"AV-66.03"(LOCK := #"lock 4",   // "Valve"
               LIOP_SEL := #init,
               L_AUT := #init,
               L_REMOTE := #init,
               L_RESET := #reset,
               AUT_OP := "BFT-66".Out_AV_Inload AND "BFT-66".InloadAV_OffTime.Q,
               L_MON := #init,
               INSTANCE := 'AV-66.03',
               QCMD_OP => "AV-66.03");
END_REGION

REGION Network 55: AV-66.04
   RUNG wire#powerrail
      #"AV-66.04"(AUT_OP := wire#w1, LOCK := #"lock 4", ERR_EXTERN :=, LIOP_SEL := #init, L_AUT := #init, L_REMOTE := #init, L_SIM :=, L_RESET := #reset, MAN_OP :=, SIM_OP :=, FB_OPEN :=, FB_CLOSE :=, L_MON := #init, MON_T :=, MON_T_CLOSE :=, INSTANCE := 'AV-66.04', RESTART :=, VISIBILITY :=, OPdwCmd :=, QdwState =>, QwState =>, QCLOSING =>, QCLOSE =>, QOPENING =>, QOPEN =>, QCMD_OP => "AV-66.04", QMON =>, QMON_ERR =>, QMON_T =>, QMON_T_CLOSE =>, QMAN_AUT =>, QREMOTE =>, QSIM =>, QLOCK =>, QERR =>, QERR_EXT =>, QwAlarm =>)
   END_RUNG
   RUNG wire#powerrail
      Contact( "BFT-66".Out_AV_CIP_Tank )
   END_RUNG wire#w1
   // the same network as SCL:
   #"AV-66.04"(LOCK := #"lock 4",   // "Valve"
               LIOP_SEL := #init,
               L_AUT := #init,
               L_REMOTE := #init,
               L_RESET := #reset,
               AUT_OP := "BFT-66".Out_AV_CIP_Tank,
               L_MON := #init,
               INSTANCE := 'AV-66.04',
               QCMD_OP => "AV-66.04");
END_REGION

REGION Network 56: AV-66.05
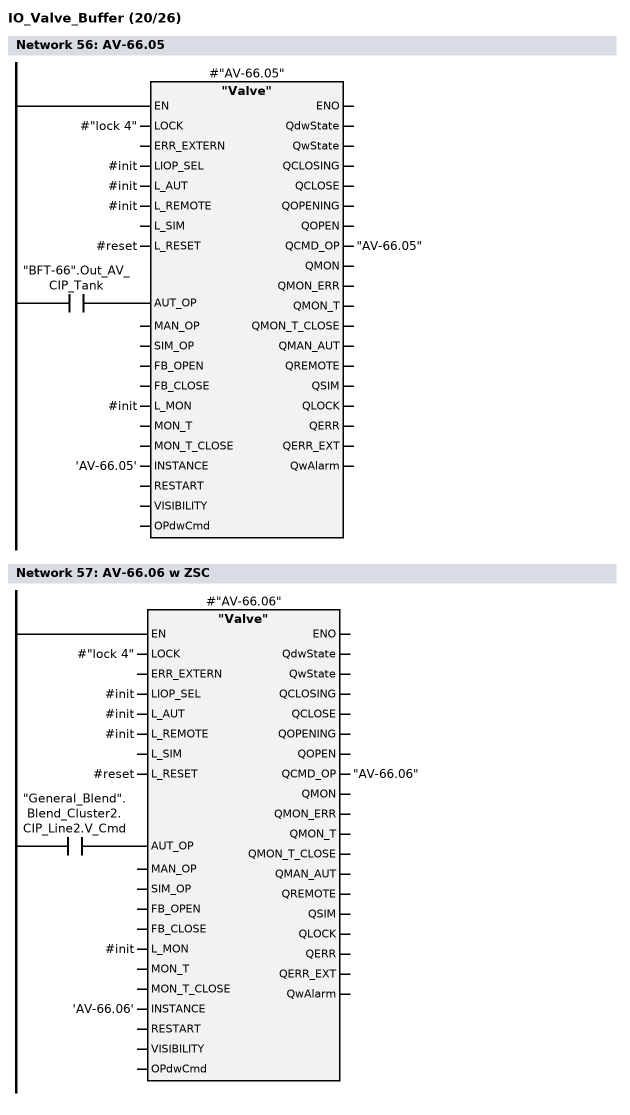
   RUNG wire#powerrail
      #"AV-66.05"(AUT_OP := wire#w1, LOCK := #"lock 4", ERR_EXTERN :=, LIOP_SEL := #init, L_AUT := #init, L_REMOTE := #init, L_SIM :=, L_RESET := #reset, MAN_OP :=, SIM_OP :=, FB_OPEN :=, FB_CLOSE :=, L_MON := #init, MON_T :=, MON_T_CLOSE :=, INSTANCE := 'AV-66.05', RESTART :=, VISIBILITY :=, OPdwCmd :=, QdwState =>, QwState =>, QCLOSING =>, QCLOSE =>, QOPENING =>, QOPEN =>, QCMD_OP => "AV-66.05", QMON =>, QMON_ERR =>, QMON_T =>, QMON_T_CLOSE =>, QMAN_AUT =>, QREMOTE =>, QSIM =>, QLOCK =>, QERR =>, QERR_EXT =>, QwAlarm =>)
   END_RUNG
   RUNG wire#powerrail
      Contact( "BFT-66".Out_AV_CIP_Tank )
   END_RUNG wire#w1
   // the same network as SCL:
   #"AV-66.05"(LOCK := #"lock 4",   // "Valve"
               LIOP_SEL := #init,
               L_AUT := #init,
               L_REMOTE := #init,
               L_RESET := #reset,
               AUT_OP := "BFT-66".Out_AV_CIP_Tank,
               L_MON := #init,
               INSTANCE := 'AV-66.05',
               QCMD_OP => "AV-66.05");
END_REGION

REGION Network 57: AV-66.06 w ZSC
   RUNG wire#powerrail
      #"AV-66.06"(AUT_OP := wire#w1, LOCK := #"lock 4", ERR_EXTERN :=, LIOP_SEL := #init, L_AUT := #init, L_REMOTE := #init, L_SIM :=, L_RESET := #reset, MAN_OP :=, SIM_OP :=, FB_OPEN :=, FB_CLOSE :=, L_MON := #init, MON_T :=, MON_T_CLOSE :=, INSTANCE := 'AV-66.06', RESTART :=, VISIBILITY :=, OPdwCmd :=, QdwState =>, QwState =>, QCLOSING =>, QCLOSE =>, QOPENING =>, QOPEN =>, QCMD_OP => "AV-66.06", QMON =>, QMON_ERR =>, QMON_T =>, QMON_T_CLOSE =>, QMAN_AUT =>, QREMOTE =>, QSIM =>, QLOCK =>, QERR =>, QERR_EXT =>, QwAlarm =>)
   END_RUNG
   RUNG wire#powerrail
      Contact( "General_Blend".Blend_Cluster2.CIP_Line2.V_Cmd )
   END_RUNG wire#w1
   // the same network as SCL:
   #"AV-66.06"(LOCK := #"lock 4",   // "Valve"
               LIOP_SEL := #init,
               L_AUT := #init,
               L_REMOTE := #init,
               L_RESET := #reset,
               AUT_OP := "General_Blend".Blend_Cluster2.CIP_Line2.V_Cmd,
               L_MON := #init,
               INSTANCE := 'AV-66.06',
               QCMD_OP => "AV-66.06");
END_REGION

REGION Network 59 (SCL): FB OPEN AND CLOSE VALVE T-67
   IF #testing THEN
       // Statement section IF
       #"AV-67.01".FB_OPEN := #"AV-67.01".QCMD_OP;
       #"AV-67.01".FB_CLOSE := NOT #"AV-67.01".QCMD_OP;
       #"AV-67.02".FB_OPEN := #"AV-67.02".QCMD_OP;
       #"AV-67.02".FB_CLOSE := NOT #"AV-67.02".QCMD_OP;
       #"AV-67.03".FB_OPEN := #"AV-67.03".QCMD_OP;
       #"AV-67.03".FB_CLOSE := NOT #"AV-67.03".QCMD_OP;
       #"AV-67.04".FB_OPEN := #"AV-67.04".QCMD_OP;
       #"AV-67.04".FB_CLOSE := NOT #"AV-67.04".QCMD_OP;
       #"AV-67.05".FB_OPEN := #"AV-67.05".QCMD_OP;
       #"AV-67.05".FB_CLOSE := NOT #"AV-67.05".QCMD_OP;
   ELSE
       // Statement section ELSE
       #"AV-67.01".FB_OPEN := NOT "ZSC-67.01";
       #"AV-67.01".FB_CLOSE := "ZSC-67.01";
       #"AV-67.02".FB_OPEN := #"AV-67.02".QCMD_OP;
       #"AV-67.02".FB_CLOSE := NOT #"AV-67.02".QCMD_OP;
       #"AV-67.03".FB_OPEN := NOT "ZSC-67.03";
       #"AV-67.03".FB_CLOSE := "ZSC-67.03";
       #"AV-67.04".FB_OPEN := #"AV-67.04".QCMD_OP;
       #"AV-67.04".FB_CLOSE := NOT #"AV-67.04".QCMD_OP;
       #"AV-67.05".FB_OPEN := #"AV-67.05".QCMD_OP;
       #"AV-67.05".FB_CLOSE := NOT #"AV-67.05".QCMD_OP;
   END_IF;
END_REGION

NETWORK
TITLE = FB MONITORING TIME VALVE T-67
// FB OPEN TIME
      L     T#20s;
      T     #"AV-67.01".MON_T;
      T     #"AV-67.02".MON_T;
      T     #"AV-67.03".MON_T;
      T     #"AV-67.04".MON_T;
      T     #"AV-67.05".MON_T;
// FB CLOSE TIME
      L     T#20s;
      T     #"AV-67.01".MON_T_CLOSE;
      T     #"AV-67.02".MON_T_CLOSE;
      T     #"AV-67.03".MON_T_CLOSE;
      T     #"AV-67.04".MON_T_CLOSE;
      T     #"AV-67.05".MON_T_CLOSE;


REGION Network 61: AV-67.01 w ZSC
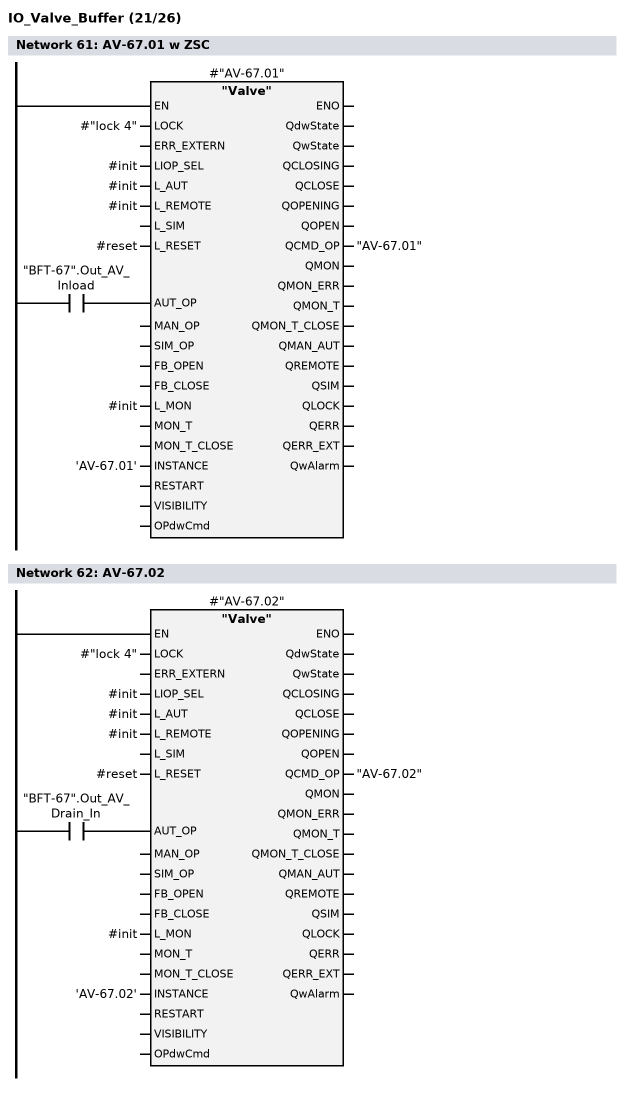
   RUNG wire#powerrail
      #"AV-67.01"(AUT_OP := wire#w1, LOCK := #"lock 4", ERR_EXTERN :=, LIOP_SEL := #init, L_AUT := #init, L_REMOTE := #init, L_SIM :=, L_RESET := #reset, MAN_OP :=, SIM_OP :=, FB_OPEN :=, FB_CLOSE :=, L_MON := #init, MON_T :=, MON_T_CLOSE :=, INSTANCE := 'AV-67.01', RESTART :=, VISIBILITY :=, OPdwCmd :=, QdwState =>, QwState =>, QCLOSING =>, QCLOSE =>, QOPENING =>, QOPEN =>, QCMD_OP => "AV-67.01", QMON =>, QMON_ERR =>, QMON_T =>, QMON_T_CLOSE =>, QMAN_AUT =>, QREMOTE =>, QSIM =>, QLOCK =>, QERR =>, QERR_EXT =>, QwAlarm =>)
   END_RUNG
   RUNG wire#powerrail
      Contact( "BFT-67".Out_AV_Inload )
   END_RUNG wire#w1
   // the same network as SCL:
   #"AV-67.01"(LOCK := #"lock 4",   // "Valve"
               LIOP_SEL := #init,
               L_AUT := #init,
               L_REMOTE := #init,
               L_RESET := #reset,
               AUT_OP := "BFT-67".Out_AV_Inload,
               L_MON := #init,
               INSTANCE := 'AV-67.01',
               QCMD_OP => "AV-67.01");
END_REGION

REGION Network 62: AV-67.02
   RUNG wire#powerrail
      #"AV-67.02"(AUT_OP := wire#w1, LOCK := #"lock 4", ERR_EXTERN :=, LIOP_SEL := #init, L_AUT := #init, L_REMOTE := #init, L_SIM :=, L_RESET := #reset, MAN_OP :=, SIM_OP :=, FB_OPEN :=, FB_CLOSE :=, L_MON := #init, MON_T :=, MON_T_CLOSE :=, INSTANCE := 'AV-67.02', RESTART :=, VISIBILITY :=, OPdwCmd :=, QdwState =>, QwState =>, QCLOSING =>, QCLOSE =>, QOPENING =>, QOPEN =>, QCMD_OP => "AV-67.02", QMON =>, QMON_ERR =>, QMON_T =>, QMON_T_CLOSE =>, QMAN_AUT =>, QREMOTE =>, QSIM =>, QLOCK =>, QERR =>, QERR_EXT =>, QwAlarm =>)
   END_RUNG
   RUNG wire#powerrail
      Contact( "BFT-67".Out_AV_Drain_In )
   END_RUNG wire#w1
   // the same network as SCL:
   #"AV-67.02"(LOCK := #"lock 4",   // "Valve"
               LIOP_SEL := #init,
               L_AUT := #init,
               L_REMOTE := #init,
               L_RESET := #reset,
               AUT_OP := "BFT-67".Out_AV_Drain_In,
               L_MON := #init,
               INSTANCE := 'AV-67.02',
               QCMD_OP => "AV-67.02");
END_REGION

REGION Network 63: AV-67.03 w ZSC
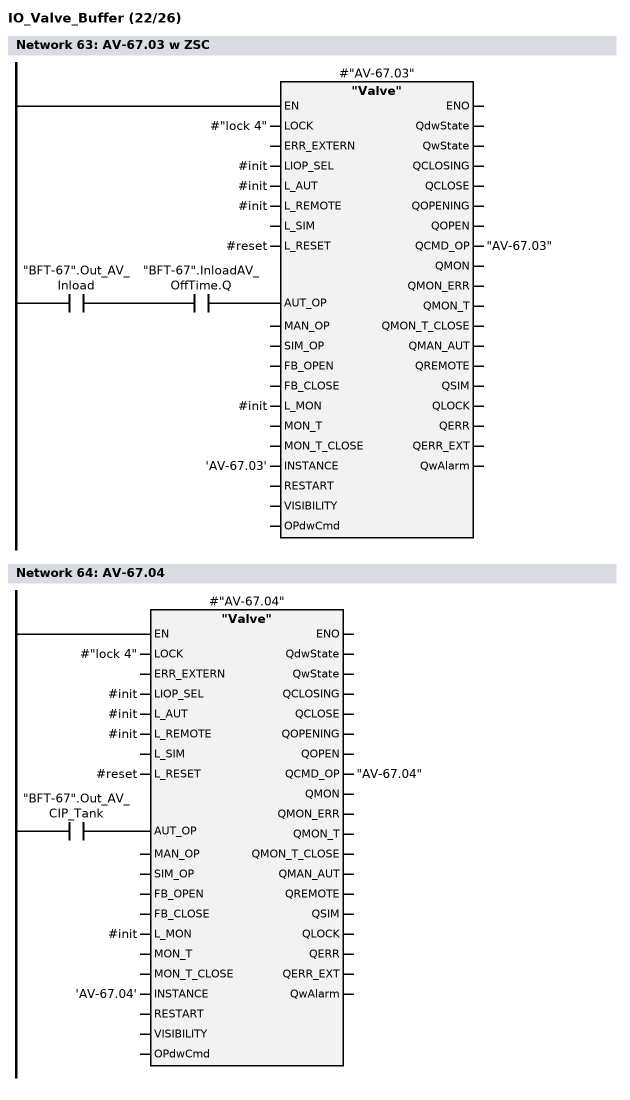
   RUNG wire#powerrail
      #"AV-67.03"(AUT_OP := wire#w1, LOCK := #"lock 4", ERR_EXTERN :=, LIOP_SEL := #init, L_AUT := #init, L_REMOTE := #init, L_SIM :=, L_RESET := #reset, MAN_OP :=, SIM_OP :=, FB_OPEN :=, FB_CLOSE :=, L_MON := #init, MON_T :=, MON_T_CLOSE :=, INSTANCE := 'AV-67.03', RESTART :=, VISIBILITY :=, OPdwCmd :=, QdwState =>, QwState =>, QCLOSING =>, QCLOSE =>, QOPENING =>, QOPEN =>, QCMD_OP => "AV-67.03", QMON =>, QMON_ERR =>, QMON_T =>, QMON_T_CLOSE =>, QMAN_AUT =>, QREMOTE =>, QSIM =>, QLOCK =>, QERR =>, QERR_EXT =>, QwAlarm =>)
   END_RUNG
   RUNG wire#powerrail
      Contact( "BFT-67".Out_AV_Inload )
      Contact( "BFT-67".InloadAV_OffTime.Q )
   END_RUNG wire#w1
   // the same network as SCL:
   #"AV-67.03"(LOCK := #"lock 4",   // "Valve"
               LIOP_SEL := #init,
               L_AUT := #init,
               L_REMOTE := #init,
               L_RESET := #reset,
               AUT_OP := "BFT-67".Out_AV_Inload AND "BFT-67".InloadAV_OffTime.Q,
               L_MON := #init,
               INSTANCE := 'AV-67.03',
               QCMD_OP => "AV-67.03");
END_REGION

REGION Network 64: AV-67.04
   RUNG wire#powerrail
      #"AV-67.04"(AUT_OP := wire#w1, LOCK := #"lock 4", ERR_EXTERN :=, LIOP_SEL := #init, L_AUT := #init, L_REMOTE := #init, L_SIM :=, L_RESET := #reset, MAN_OP :=, SIM_OP :=, FB_OPEN :=, FB_CLOSE :=, L_MON := #init, MON_T :=, MON_T_CLOSE :=, INSTANCE := 'AV-67.04', RESTART :=, VISIBILITY :=, OPdwCmd :=, QdwState =>, QwState =>, QCLOSING =>, QCLOSE =>, QOPENING =>, QOPEN =>, QCMD_OP => "AV-67.04", QMON =>, QMON_ERR =>, QMON_T =>, QMON_T_CLOSE =>, QMAN_AUT =>, QREMOTE =>, QSIM =>, QLOCK =>, QERR =>, QERR_EXT =>, QwAlarm =>)
   END_RUNG
   RUNG wire#powerrail
      Contact( "BFT-67".Out_AV_CIP_Tank )
   END_RUNG wire#w1
   // the same network as SCL:
   #"AV-67.04"(LOCK := #"lock 4",   // "Valve"
               LIOP_SEL := #init,
               L_AUT := #init,
               L_REMOTE := #init,
               L_RESET := #reset,
               AUT_OP := "BFT-67".Out_AV_CIP_Tank,
               L_MON := #init,
               INSTANCE := 'AV-67.04',
               QCMD_OP => "AV-67.04");
END_REGION

REGION Network 65: AV-67.05
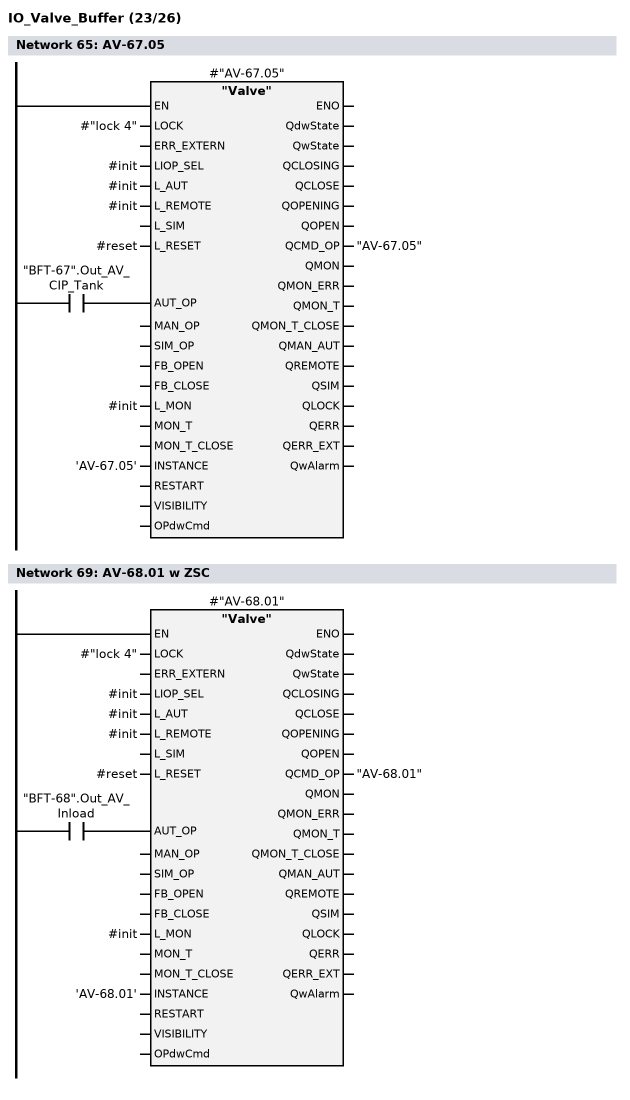
   RUNG wire#powerrail
      #"AV-67.05"(AUT_OP := wire#w1, LOCK := #"lock 4", ERR_EXTERN :=, LIOP_SEL := #init, L_AUT := #init, L_REMOTE := #init, L_SIM :=, L_RESET := #reset, MAN_OP :=, SIM_OP :=, FB_OPEN :=, FB_CLOSE :=, L_MON := #init, MON_T :=, MON_T_CLOSE :=, INSTANCE := 'AV-67.05', RESTART :=, VISIBILITY :=, OPdwCmd :=, QdwState =>, QwState =>, QCLOSING =>, QCLOSE =>, QOPENING =>, QOPEN =>, QCMD_OP => "AV-67.05", QMON =>, QMON_ERR =>, QMON_T =>, QMON_T_CLOSE =>, QMAN_AUT =>, QREMOTE =>, QSIM =>, QLOCK =>, QERR =>, QERR_EXT =>, QwAlarm =>)
   END_RUNG
   RUNG wire#powerrail
      Contact( "BFT-67".Out_AV_CIP_Tank )
   END_RUNG wire#w1
   // the same network as SCL:
   #"AV-67.05"(LOCK := #"lock 4",   // "Valve"
               LIOP_SEL := #init,
               L_AUT := #init,
               L_REMOTE := #init,
               L_RESET := #reset,
               AUT_OP := "BFT-67".Out_AV_CIP_Tank,
               L_MON := #init,
               INSTANCE := 'AV-67.05',
               QCMD_OP => "AV-67.05");
END_REGION

REGION Network 67 (SCL): FB OPEN AND CLOSE VALVE T-68
   IF #testing THEN
       // Statement section IF
       #"AV-68.01".FB_OPEN := #"AV-68.01".QCMD_OP;
       #"AV-68.01".FB_CLOSE := NOT #"AV-68.01".QCMD_OP;
       #"AV-68.02".FB_OPEN := #"AV-68.02".QCMD_OP;
       #"AV-68.02".FB_CLOSE := NOT #"AV-68.02".QCMD_OP;
       #"AV-68.03".FB_OPEN := #"AV-68.03".QCMD_OP;
       #"AV-68.03".FB_CLOSE := NOT #"AV-68.03".QCMD_OP;
       #"AV-68.04".FB_OPEN := #"AV-68.04".QCMD_OP;
       #"AV-68.04".FB_CLOSE := NOT #"AV-68.04".QCMD_OP;
       #"AV-68.05".FB_OPEN := #"AV-68.05".QCMD_OP;
       #"AV-68.05".FB_CLOSE := NOT #"AV-68.05".QCMD_OP;
       #"AV-68.06".FB_OPEN := #"AV-68.06".QCMD_OP;
       #"AV-68.06".FB_CLOSE := NOT #"AV-68.06".QCMD_OP;
   ELSE
       // Statement section ELSE
       #"AV-68.01".FB_OPEN := NOT "ZSC-68.01";
       #"AV-68.01".FB_CLOSE := "ZSC-68.01";
       #"AV-68.02".FB_OPEN := #"AV-68.02".QCMD_OP;
       #"AV-68.02".FB_CLOSE := NOT #"AV-68.02".QCMD_OP;
       #"AV-68.03".FB_OPEN := NOT "ZSC-68.03";
       #"AV-68.03".FB_CLOSE := "ZSC-68.03";
       #"AV-68.04".FB_OPEN := #"AV-68.04".QCMD_OP;
       #"AV-68.04".FB_CLOSE := NOT #"AV-68.04".QCMD_OP;
       #"AV-68.05".FB_OPEN := #"AV-68.05".QCMD_OP;
       #"AV-68.05".FB_CLOSE := NOT #"AV-68.05".QCMD_OP;
       #"AV-68.06".FB_OPEN := NOT "ZSC-68.06";
       #"AV-68.06".FB_CLOSE := "ZSC-68.06";
   END_IF;
END_REGION

NETWORK
TITLE = FB MONITORING TIME VALVE T-68
// FB OPEN TIME
      L     T#20s;
      T     #"AV-68.01".MON_T;
      T     #"AV-68.02".MON_T;
      T     #"AV-68.03".MON_T;
      T     #"AV-68.04".MON_T;
      T     #"AV-68.05".MON_T;
      T     #"AV-68.06".MON_T;
// FB CLOSE TIME
      L     T#20s;
      T     #"AV-68.01".MON_T_CLOSE;
      T     #"AV-68.02".MON_T_CLOSE;
      T     #"AV-68.03".MON_T_CLOSE;
      T     #"AV-68.04".MON_T_CLOSE;
      T     #"AV-68.05".MON_T_CLOSE;
      T     #"AV-68.06".MON_T_CLOSE;

REGION Network 69: AV-68.01 w ZSC
   RUNG wire#powerrail
      #"AV-68.01"(AUT_OP := wire#w1, LOCK := #"lock 4", ERR_EXTERN :=, LIOP_SEL := #init, L_AUT := #init, L_REMOTE := #init, L_SIM :=, L_RESET := #reset, MAN_OP :=, SIM_OP :=, FB_OPEN :=, FB_CLOSE :=, L_MON := #init, MON_T :=, MON_T_CLOSE :=, INSTANCE := 'AV-68.01', RESTART :=, VISIBILITY :=, OPdwCmd :=, QdwState =>, QwState =>, QCLOSING =>, QCLOSE =>, QOPENING =>, QOPEN =>, QCMD_OP => "AV-68.01", QMON =>, QMON_ERR =>, QMON_T =>, QMON_T_CLOSE =>, QMAN_AUT =>, QREMOTE =>, QSIM =>, QLOCK =>, QERR =>, QERR_EXT =>, QwAlarm =>)
   END_RUNG
   RUNG wire#powerrail
      Contact( "BFT-68".Out_AV_Inload )
   END_RUNG wire#w1
   // the same network as SCL:
   #"AV-68.01"(LOCK := #"lock 4",   // "Valve"
               LIOP_SEL := #init,
               L_AUT := #init,
               L_REMOTE := #init,
               L_RESET := #reset,
               AUT_OP := "BFT-68".Out_AV_Inload,
               L_MON := #init,
               INSTANCE := 'AV-68.01',
               QCMD_OP => "AV-68.01");
END_REGION

REGION Network 70: AV-68.02
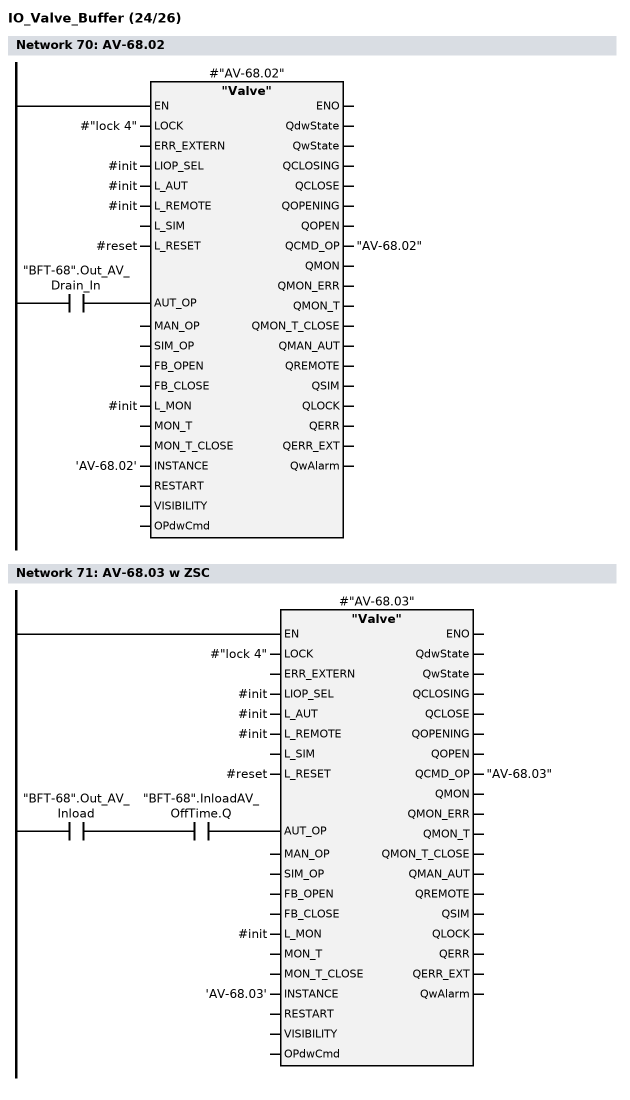
   RUNG wire#powerrail
      #"AV-68.02"(AUT_OP := wire#w1, LOCK := #"lock 4", ERR_EXTERN :=, LIOP_SEL := #init, L_AUT := #init, L_REMOTE := #init, L_SIM :=, L_RESET := #reset, MAN_OP :=, SIM_OP :=, FB_OPEN :=, FB_CLOSE :=, L_MON := #init, MON_T :=, MON_T_CLOSE :=, INSTANCE := 'AV-68.02', RESTART :=, VISIBILITY :=, OPdwCmd :=, QdwState =>, QwState =>, QCLOSING =>, QCLOSE =>, QOPENING =>, QOPEN =>, QCMD_OP => "AV-68.02", QMON =>, QMON_ERR =>, QMON_T =>, QMON_T_CLOSE =>, QMAN_AUT =>, QREMOTE =>, QSIM =>, QLOCK =>, QERR =>, QERR_EXT =>, QwAlarm =>)
   END_RUNG
   RUNG wire#powerrail
      Contact( "BFT-68".Out_AV_Drain_In )
   END_RUNG wire#w1
   // the same network as SCL:
   #"AV-68.02"(LOCK := #"lock 4",   // "Valve"
               LIOP_SEL := #init,
               L_AUT := #init,
               L_REMOTE := #init,
               L_RESET := #reset,
               AUT_OP := "BFT-68".Out_AV_Drain_In,
               L_MON := #init,
               INSTANCE := 'AV-68.02',
               QCMD_OP => "AV-68.02");
END_REGION

REGION Network 71: AV-68.03 w ZSC
   RUNG wire#powerrail
      #"AV-68.03"(AUT_OP := wire#w1, LOCK := #"lock 4", ERR_EXTERN :=, LIOP_SEL := #init, L_AUT := #init, L_REMOTE := #init, L_SIM :=, L_RESET := #reset, MAN_OP :=, SIM_OP :=, FB_OPEN :=, FB_CLOSE :=, L_MON := #init, MON_T :=, MON_T_CLOSE :=, INSTANCE := 'AV-68.03', RESTART :=, VISIBILITY :=, OPdwCmd :=, QdwState =>, QwState =>, QCLOSING =>, QCLOSE =>, QOPENING =>, QOPEN =>, QCMD_OP => "AV-68.03", QMON =>, QMON_ERR =>, QMON_T =>, QMON_T_CLOSE =>, QMAN_AUT =>, QREMOTE =>, QSIM =>, QLOCK =>, QERR =>, QERR_EXT =>, QwAlarm =>)
   END_RUNG
   RUNG wire#powerrail
      Contact( "BFT-68".Out_AV_Inload )
      Contact( "BFT-68".InloadAV_OffTime.Q )
   END_RUNG wire#w1
   // the same network as SCL:
   #"AV-68.03"(LOCK := #"lock 4",   // "Valve"
               LIOP_SEL := #init,
               L_AUT := #init,
               L_REMOTE := #init,
               L_RESET := #reset,
               AUT_OP := "BFT-68".Out_AV_Inload AND "BFT-68".InloadAV_OffTime.Q,
               L_MON := #init,
               INSTANCE := 'AV-68.03',
               QCMD_OP => "AV-68.03");
END_REGION

REGION Network 72: AV-68.04
